Omron CX-Programmer project NewProject (CX-Programmer 9.74)

# PLC MES_Trat: CJ2M CPU34
I/O table (CPU CJ2M-CPU34): rack 0 slot 0 CJ1W-OD232; rack 0 slot 11 CJ2M-EIP21

## Data types
TYPE Evento : STRUCT
  Ciclo : BOOL;  (* Em Ciclo Produtivo PLC->MES *)
  Estado : INT;  (* Estado Equipamento PLC->MES *)
  EquiDesabil : BOOL Dimensions=[16];  (* Equipamento Desabilitado PLC->MES *)
  FimCiclo : BOOL;  (* Finalização Ciclo PLC->MES *)
END_STRUCT END_TYPE
TYPE Ordem_Cmd : STRUCT
  AutoMES : BOOL;  (* Autorização MES MES->PLC *)
  QtdFaltaOF : UDINT;  (* Quantidade Em Falta OF *)
  ProdExecMaquina : UDINT;  (* Produção Executada Máquina *)
END_STRUCT END_TYPE
TYPE Ordem : STRUCT
  Ordem : DINT;  (* OF_OM MES->PLC *)
  Sinalizacao : BOOL;
  ProdExpect : UDINT;  (* Produção Expectável MES->PLC *)
  ProdExecOrdem : UDINT;  (* Produção Executada Ordem MES->PLC *)
END_STRUCT END_TYPE
TYPE InfoAux : STRUCT
  Cliente : WORD Dimensions=[50];  (* Cliente (string) MES->PLC *)
  Artigo : WORD Dimensions=[50];  (* Artigo (string) MES->PLC *)
  Encomenda : WORD Dimensions=[50];  (* Encomenda (string) MES->PLC *)
  QtdEncom : UDINT;  (* Quantidade Encomenda MES->PLC *)
  QtdReal : UDINT;  (* Quantidade Real MES->PLC *)
  NomeReceita : WORD Dimensions=[50];  (* Nome Receita (string) MES->PLC *)
  DataExpedic : WORD Dimensions=[4];  (* Data Expedição (string) MES->PLC *)
END_STRUCT END_TYPE
TYPE BStep : STRUCT  (* Batch Load/Exec Steps defenition *)
  Func : DWORD;  (* Function *)
  Param01 : DWORD;
  Param02 : DWORD;
END_STRUCT END_TYPE
TYPE BatchLoad : STRUCT
  InfoAux : InfoAux;
  Ordem : DINT;  (* Ordem MES->PLC *)
  Chk : WORD;  (* CheckSum MES->PLC *)
  Steps : BStep Dimensions=[12];  (* Steps MES->PLC *)
END_STRUCT END_TYPE
TYPE BatchExec : STRUCT
  Steps : BStep Dimensions=[12];  (* PLC->MES *)
END_STRUCT END_TYPE
TYPE RStep : STRUCT  (* Batch Real Step defenition *)
  Active : BOOL;
  Value01 : DWORD;
  Value02 : DWORD;
END_STRUCT END_TYPE
TYPE BatchReal : STRUCT
  Heat : RStep;  (* PLC->MES *)
  Inje : RStep;  (* PLC->MES *)
  Dedu : RStep;  (* PLC->MES *)
  Tumb : RStep;  (* PLC->MES *)
  Load : RStep;  (* PLC->MES *)
  Unload : RStep;  (* PLC->MES *)
END_STRUCT END_TYPE
TYPE s_of_totais : STRUCT  (* Totais produzidos e a produzir de uma OF *)
  tt_global : UDINT;  (* Total a produzir na OF *)
  tt_falta : UDINT;  (* Total que falta produzir na OF *)
  tt_produzir : UDINT;  (* Total a produzir na maquina no batch *)
  tt_cestos : UDINT;  (* Total de cestos a produzir na OF *)
END_STRUCT END_TYPE
TYPE s_of_cliente : STRUCT  (* Dados do cliente de uma OF *)
  Cliente : WORD Dimensions=[50];
  Artigo : WORD Dimensions=[50];
  Encomenda : WORD Dimensions=[50];
  QtdEncomenda : UDINT;
  QtdReal : UDINT;
  DataExpedicao : WORD Dimensions=[4];
  NomeReceita : WORD Dimensions=[50];
  nome : WORD Dimensions=[25];
  data : WORD Dimensions=[10];
  produto : WORD Dimensions=[20];
  prg_on : WORD Dimensions=[5];
  n_enc : WORD Dimensions=[10];
  n_of : WORD Dimensions=[10];
  n_lt : WORD Dimensions=[10];
  rsv2 : INT Dimensions=[10];
END_STRUCT END_TYPE
TYPE s_of_pss : STRUCT  (* Passo individual do programa a executar *)
  f : INT;  (* Função *)
  p1 : INT;  (* Parametro 1 *)
  p2 : REAL;  (* Parametro 2 *)
  tt : REAL;  (* Totalizador *)
  uni : INT;  (* Unidade *)
  b0 : BOOL;  (* Bit - É função *)
  b1 : BOOL;  (* Bit - É produto *)
  b2 : BOOL;  (* Bit - Tem tempo *)
  b3 : BOOL;  (* Bit - Tem quantidade *)
  b4 : BOOL;  (* Bit - Tem temperatura *)
  tt_inv : REAL;  (* Contagem Inversa *)
END_STRUCT END_TYPE
TYPE s_of_prg : STRUCT  (* Programa a ser executado *)
  pss : s_of_pss Dimensions=[12];  (* Passos do programa a executar *)
END_STRUCT END_TYPE
TYPE s_of : STRUCT  (* Ordem de fabrico *)
  cliente : s_of_cliente;  (* Cliente da OF *)
  totais : s_of_totais;  (* Totais da OF *)
  dados : BOOL;  (* OF com valores *)
  online : BOOL;  (* Ordem com dados para funcionar online *)
  rep : BOOL;  (* OF/Lote reprocessado *)
  of_del : BOOL;  (* Apagar OF *)
  sel_cestos_rolhas : BOOL;  (* Botão de Selecção entre inserção de número de rolhas e número de cestos a produzir *)
  nprg_off : INT;  (* Numero do programa offline *)
  prg : s_of_prg;  (* Programa *)
END_STRUCT END_TYPE
TYPE Passos : STRUCT
  f : INT;
  p1 : INT;
  p2 : REAL;
END_STRUCT END_TYPE
TYPE ReceitaMaq : STRUCT
  Step : Passos Dimensions=[12];
END_STRUCT END_TYPE
TYPE s_Steps : STRUCT
  f : INT;  (* Função *)
  p1 : INT;  (* Parametro 1 *)
  p2 : REAL;  (* Parametro 2 *)
END_STRUCT END_TYPE
TYPE s_Step : STRUCT
  f : INT;  (* Função *)
  p1 : INT;  (* Parametro 1 *)
  p2 : REAL;  (* Parametro 2 *)
  No : INT;  (* Numero do Passo *)
END_STRUCT END_TYPE
TYPE s_Estado : STRUCT
  Ciclo : BOOL;  (* Em ciclo produtivo *)
  FimCiclo : BOOL;  (* Finalização ciclo *)
  Estado : BOOL;  (* Estado equipamento *)
  FimTratamento : BOOL;  (* Tratamento Finalizado *)
  OF_Carregada : BOOL;  (* Ordem carregada para máquina *)
  Avaria : BOOL;  (* Máquina em Avaria *)
  Com_OF : BOOL;  (* Máquina com OF carregada *)
  FalhaInjeProd : BOOL;  (* Falta de injeção de produto *)
  FalhaAquecim : BOOL;  (* Falha de aquecimento *)
  AvariaTermicos : BOOL;  (* Avaria de térmicos *)
  TratAbortado : BOOL;  (* Tratamento abortado pelo operador *)
  FalhaEnergia : BOOL;  (* Falha energia *)
  NivelProdBaixo : BOOL;  (* Nível produto químico no depósito baixo *)
  Manual : BOOL;  (* modo manual *)
  Emergencia : BOOL;  (* Paragem Emergência *)
END_STRUCT END_TYPE
TYPE s_produtos : STRUCT
  CodMES : WORD Dimensions=[4];
  CodPLC : INT;
END_STRUCT END_TYPE
TYPE M1_Param : STRUCT  (* Parametros do passo *)
  Manual : BOOL;  (* Espera por confirmação manual do operador *)
  Auto : BOOL;  (* Avança automáticamente *)
  P1 : BOOL;  (* Produto 1 *)
  P2 : BOOL;  (* Produto 2 *)
  P3 : BOOL;  (* Produto 3 *)
  P4 : BOOL;  (* Produto 4 *)
  DEDU : BOOL;  (* Asperação (Blower) *)
  HEAT : BOOL;  (* Aquecimento (Heater) *)
  TUMB : BOOL;  (* Rotação (Speed) *)
  LOAD : BOOL;  (* Carga *)
  UNLO : BOOL;  (* Descarga (unload) *)
  Reserva : BOOL;
  End : BOOL;
  CalTemp : BOOL;  (* Calor por Temperatura *)
  Cool : BOOL;  (* Arrefecimento *)
END_STRUCT END_TYPE
TYPE M1_ParamProd : STRUCT  (* Parametros produtos *)
  DoseRate : BOOL;  (* por Dosagem g/m *)
  Qtd : BOOL;  (* por Quantidade q *)
  Time : BOOL;  (* poe Tempo mm:ss *)
  Cycles : BOOL;  (* por Ciclos *)
END_STRUCT END_TYPE
TYPE M1_Step : STRUCT  (* Passo da Receita *)
  Parametros : M1_Param;  (* Parametros do Passo *)
  ParamProdutos : M1_ParamProd Dimensions=[4];
  Temperatura : INT;  (* Valor da Temperatura *)
  Velocidade : INT;  (* Valor Velocidade Rotação (%) *)
  P1 : INT;  (* Valor Produto 1 *)
  P2 : INT;  (* Valor Produto 2 *)
  P3 : INT;  (* Valor Produto 3 *)
  P4 : BOOL;  (* Valor do Produto 4 *)
  Tempo : BOOL;  (* Tempo (mm:ss) *)
  Reserva : INT;
  P1_TOff_TOn : INT;  (* TOff/TON P1 *)
  P2_TOff_TOn : INT;  (* TOff/TON P2 *)
  P3_TOff_TOn : INT;  (* TOff/TON P3 *)
  P4_TOff_TOn : INT;  (* TOff/TON P4 *)
END_STRUCT END_TYPE
TYPE s_Controlo : STRUCT
  Mannual : BOOL;
  Auto : BOOL;
  P1 : BOOL;
  P2 : BOOL;
  P3 : BOOL;
  P4 : BOOL;
  Aspiracao : BOOL;
  Aquecimento : BOOL;
  Rotacao : BOOL;
  Carga : BOOL;
  Descarga : BOOL;
  Reserva1 : BOOL;
  Fim : BOOL;
  CalorPorTemperatura : BOOL;
  Arrefecimento : BOOL;
  Reserva2 : BOOL;
  Ctrl_P1 : s_CtrlProduto;
  Ctrl_P2 : s_CtrlProduto;
  Ctrl_P3 : s_CtrlProduto;
  Ctrl_P4 : BOOL;
END_STRUCT END_TYPE
TYPE s_CtrlProduto : STRUCT  (* Bits controlo produto *)
  DoseRate : BOOL;
  Qtd : BOOL;
  Time : BOOL;
  Cycles : BOOL;
END_STRUCT END_TYPE
TYPE s_StepRcpMaq1 : STRUCT  (* Receita máquina 1 *)
  Control : s_Controlo;
  Temperatura : UINT;
  Velocidade : UINT;
  ValorProduto : UINT;  (* Valor do Produto a Injetar (minutos/segundos) *)
  Tempo : UINT;  (* Tempo em segundos (minutos/segundos) *)
END_STRUCT END_TYPE
TYPE s_Evento : STRUCT
  HeartBeat : INT;  (* Heart Beat Maquina *)
  TSemHB : INT;  (* Tempo Sem Heart Beat *)
END_STRUCT END_TYPE
TYPE MqDL : STRUCT  (* 'All the mid-branches are substituted bu ".sub_Fcn."' *)
  Ordem : DINT;
  Ordem_BL : DINT;
  ProdExpect : UDINT;
  ProdEecOrdem : UDINT;
  QtdEncom : UDINT;
  QtdReal : UDINT;
  QtdEncom_BL : UDINT;
  QtdReal_BL : UDINT;
  Sinalizacao : BOOL Dimensions=[32];
  Cliente : WORD Dimensions=[50];
  Artigo : WORD Dimensions=[50];
  Encomenda : WORD Dimensions=[50];
  NomeReceita : WORD Dimensions=[50];
  Cliente_BL : WORD Dimensions=[50];
  Artigo_BL : WORD Dimensions=[50];
  Encomenda_BL : WORD Dimensions=[50];
  NomeReceita_BL : WORD Dimensions=[50];
  DataExpedic_BL : WORD Dimensions=[4];
  DataExpedic : WORD Dimensions=[4];
  Steps_BL : BStep Dimensions=[12];
END_STRUCT END_TYPE
TYPE MqRT : STRUCT  (* 'All the mid-branches are substituted bu ".sub_Fcn."' *)
  Ciclo : BOOL;
  Estado : INT;
  EquiDesabil : BOOL Dimensions=[16];
  FimCiclo : BOOL Dimensions=[16];
  AutoMes : BOOL Dimensions=[16];
  QtdFaltaOF : UDINT;
  ProExecOrdem : UDINT;
  Chk : WORD;
  Temperatura : UINT;
  BatchReal : BatchReal;
  Destination : UINT;
END_STRUCT END_TYPE

## Global symbols (name address type ; comment)
BatchReal_Maq01 E0_23050 STRUCT s_Steps
BatchReal_Maq02 E0_23150 STRUCT s_Steps
BatchReal_Maq03 E0_23250 STRUCT s_Steps
BatchReal_Maq04 E0_23350 STRUCT s_Steps
BatchReal_Maq05 E0_23450 STRUCT s_Steps
BatchReal_Maq06 E0_23550 STRUCT s_Steps
BatchReal_Maq07 E0_23650 STRUCT s_Steps
BatchReal_Maq08 E0_23750 STRUCT s_Steps
BatchReal_Maq09 E0_23850 STRUCT s_Steps
BatchReal_Maq10 E0_23950 STRUCT s_Steps
BatchReal_Maq11 E0_24050 STRUCT s_Steps
CHK_M01 D12290 WORD
CHK_M02 D12293 WORD
CHK_M03 D12296 WORD
CHK_M04 D12299 WORD
CHK_M05 D12302 WORD
CHK_M06 D12305 WORD
CHK_M07 D12308 WORD
CHK_M08 D12311 WORD
CHK_M09 D12314 WORD
CHK_M10 D12317 WORD
CHK_M11 D12320 WORD
CopyStps CopySteps
CopyStps09 CopySteps
CopyStps10 CopySteps
CopyStps11 CopySteps
CopyStps2 CopySteps
CopyStps3 CopySteps
CopyStps4 CopySteps
CopyStps5 CopySteps
CopyStps6 CopySteps
CopyStps7 CopySteps
CopyStps8 CopySteps
Estado_Maq01 E0_23057 STRUCT s_Estado
Estado_Maq02 E0_23157 STRUCT s_Estado
Estado_Maq03 E0_23257 STRUCT s_Estado
Estado_Maq04 E0_23357 STRUCT s_Estado
Estado_Maq05 E0_23457 STRUCT s_Estado
Estado_Maq06 E0_23557 STRUCT s_Estado
Estado_Maq07 E0_23657 STRUCT s_Estado
Estado_Maq08 E0_23757 STRUCT s_Estado
Estado_Maq09 E0_23857 STRUCT s_Estado
Estado_Maq10 E0_23957 STRUCT s_Estado
Estado_Maq11 E0_24057 STRUCT s_Estado
HB_M01 D12288 INT
HB_M02 D12291 INT
HB_M03 D12294 INT
HB_M04 D12297 INT
HB_M05 D12300 INT
HB_M06 D12303 INT
HB_M07 D12306 INT
HB_M08 D12309 INT
HB_M09 D12312 INT
HB_M10 D12315 INT
HB_M11 D12318 INT
M1_Tsfr_Rqst E0_25100.00 BOOL
M2_Tsfr_Rqst E0_25100.01 BOOL
M3_Tsfr_Rqst E0_25100.02 BOOL
M4_Tsfr_Rqst E0_25100.03 BOOL
M5_Tsfr_Rqst E0_25100.04 BOOL
M6_Tsfr_Rqst E0_25100.05 BOOL
MQ01_InfoAuxMq D15000 STRUCT InfoAux  ; InfoAux da receita na máquina
MQ02_InfoAuxMq D15250 STRUCT InfoAux  ; InfoAux da receita na máquina
MQ03_InfoAuxMq D15500 STRUCT InfoAux  ; InfoAux da receita na máquina
MQ04_InfoAuxMq D15750 STRUCT InfoAux  ; InfoAux da receita na máquina
MQ05_InfoAuxMq D16000 STRUCT InfoAux  ; InfoAux da receita na máquina
MQ06_InfoAuxMq D16250 STRUCT InfoAux  ; InfoAux da receita na máquina
MQ07_InfoAuxMq D16500 STRUCT InfoAux  ; InfoAux da receita na máquina
MQ08_InfoAuxMq D16750 STRUCT InfoAux  ; InfoAux da receita na máquina
MQ09_InfoAuxMq D17000 STRUCT InfoAux  ; InfoAux da receita na máquina
MQ10_InfoAuxMq D17250 STRUCT InfoAux  ; InfoAux da receita na máquina
MQ11_InfoAuxMq D17500 STRUCT InfoAux  ; InfoAux da receita na máquina
MaqDL_01 D5120 STRUCT MqDL
MaqDL_02 D5618 STRUCT MqDL
MaqDL_03 D6116 STRUCT MqDL
MaqDL_04 D6614 STRUCT MqDL
MaqDL_05 D7112 STRUCT MqDL
MaqDL_06 D7610 STRUCT MqDL
MaqDL_07 D8108 STRUCT MqDL
MaqDL_08 D8606 STRUCT MqDL
MaqDL_09 D9104 STRUCT MqDL
MaqDL_10 D9602 STRUCT MqDL
MaqDL_11 D10100 STRUCT MqDL
MaqRT_01 D0 STRUCT MqRT
MaqRT_02 D42 STRUCT MqRT
MaqRT_03 D84 STRUCT MqRT
MaqRT_04 D126 STRUCT MqRT
MaqRT_05 D168 STRUCT MqRT
MaqRT_06 D210 STRUCT MqRT
MaqRT_07 D252 STRUCT MqRT
MaqRT_08 D294 STRUCT MqRT
MaqRT_09 D336 STRUCT MqRT
MaqRT_10 D378 STRUCT MqRT
MaqRT_11 D420 STRUCT MqRT
MaqRcpNetIN_01 E0_10000 STRUCT s_of
MaqRcpNetIN_02 E0_11000 STRUCT s_of
MaqRcpNetIN_03 E0_12000 STRUCT s_of
MaqRcpNetIN_04 E0_13000 STRUCT s_of
MaqRcpNetIN_05 E0_14000 STRUCT s_of
MaqRcpNetIN_06 E0_15000 STRUCT s_of
MaqRcpNetIN_07 E0_16000 STRUCT s_of
MaqRcpNetIN_08 E0_17000 STRUCT s_of
MaqRcpNetIN_09 E0_18000 STRUCT s_of
MaqRcpNetIN_10 E0_19000 STRUCT s_of
MaqRcpNetIN_11 E0_20000 STRUCT s_of
MaqRcpNet_01 E0_0 STRUCT s_of
MaqRcpNet_02 E0_1000 STRUCT s_of
MaqRcpNet_03 E0_2000 STRUCT s_of
MaqRcpNet_04 E0_3000 STRUCT s_of
MaqRcpNet_05 E0_4000 STRUCT s_of
MaqRcpNet_06 E0_5000 STRUCT s_of
MaqRcpNet_07 E0_6000 STRUCT s_of
MaqRcpNet_08 E0_7000 STRUCT s_of
MaqRcpNet_09 E0_8000 STRUCT s_of
MaqRcpNet_10 E0_9000 STRUCT s_of
MaqRcpNet_11 E0_21000 STRUCT s_of
Mq09_CRC_Calc RecipeCRC
Mq10_CRC_Calc RecipeCRC
Mq11_CRC_Calc RecipeCRC
Mq1_CRC_Calc RecipeCRC
Mq2_CRC_Calc RecipeCRC
Mq3_CRC_Calc RecipeCRC
Mq4_CRC_Calc RecipeCRC
Mq5_CRC_Calc RecipeCRC
Mq6_CRC_Calc RecipeCRC
Mq7_CRC_Calc RecipeCRC
Mq8_CRC_Calc RecipeCRC
PLC_MES PLC_to_MES
PLC_MES09 PLC_to_MES
PLC_MES10 PLC_to_MES
PLC_MES11 PLC_to_MES
PLC_MES2 PLC_to_MES
PLC_MES3 PLC_to_MES
PLC_MES4 PLC_to_MES
PLC_MES5 PLC_to_MES
PLC_MES6 PLC_to_MES
PLC_MES7 PLC_to_MES
PLC_MES8 PLC_to_MES
Produtos H0 STRUCT[13] s_produtos
RcpTrans RecipeTranslate
RcpTrans09 RecipeTranslate
RcpTrans10 RecipeTranslate
RcpTrans11 RecipeTranslate
RcpTrans2 RecipeTranslate
RcpTrans3 RecipeTranslate
RcpTrans4 RecipeTranslate
RcpTrans5 RecipeTranslate
RcpTrans6 RecipeTranslate
RcpTrans7 RecipeTranslate
RcpTrans8 RecipeTranslate
RcpTst RecipeTst
RcpTst09 RecipeTst
RcpTst10 RecipeTst
RcpTst11 RecipeTst
RcpTst2 RecipeTst
RcpTst3 RecipeTst
RcpTst4 RecipeTst
RcpTst5 RecipeTst
RcpTst6 RecipeTst
RcpTst7 RecipeTst
RcpTst8 RecipeTst
ReceitaMaqOK_01 E0_23048.00 BOOL
ReceitaMaqOK_02 E0_23148.00 BOOL
ReceitaMaqOK_03 E0_23248.00 BOOL
ReceitaMaqOK_04 E0_23348.00 BOOL
ReceitaMaqOK_05 E0_23448.00 BOOL
ReceitaMaqOK_06 E0_23548.00 BOOL
ReceitaMaqOK_07 E0_23648.00 BOOL
ReceitaMaqOK_08 E0_23748.00 BOOL
ReceitaMaqOK_09 E0_23848.00 BOOL
ReceitaMaqOK_10 E0_23948.00 BOOL
ReceitaMaqOK_11 E0_24048.00 BOOL
ReceitaMaq_01 E0_23000 STRUCT[12] Passos
ReceitaMaq_02 E0_23100 STRUCT[12] Passos
ReceitaMaq_03 E0_23200 STRUCT[12] Passos
ReceitaMaq_04 E0_23300 STRUCT[12] Passos
ReceitaMaq_05 E0_23400 STRUCT[12] Passos
ReceitaMaq_06 E0_23500 STRUCT[12] Passos
ReceitaMaq_07 E0_23600 STRUCT[12] Passos
ReceitaMaq_08 E0_23700 STRUCT[12] Passos
ReceitaMaq_09 E0_23800 STRUCT[12] Passos
ReceitaMaq_10 E0_23900 STRUCT[12] Passos
ReceitaMaq_11 E0_24000 STRUCT[12] Passos
Send_M7 _CPU010_SendData
TSemHB_M01 D12289 INT
TSemHB_M02 D12292 INT
TSemHB_M03 D12295 INT
TSemHB_M04 D12298 INT
TSemHB_M05 D12301 INT
TSemHB_M06 D12304 INT
TSemHB_M07 D12307 INT
TSemHB_M08 D12310 INT
TSemHB_M09 D12313 INT
TSemHB_M10 D12316 INT
TSemHB_M11 D12319 INT
Teperatura_Maq01 E0_23055 INT
Teperatura_Maq02 E0_23155 INT
Teperatura_Maq03 E0_23255 INT
Teperatura_Maq04 E0_23355 INT
Teperatura_Maq05 E0_23455 INT
Teperatura_Maq06 E0_23555 INT
Teperatura_Maq07 E0_23655 INT  ; ~
Teperatura_Maq08 E0_23755 INT
Teperatura_Maq09 E0_23855 INT
Teperatura_Maq10 E0_23955 INT
Teperatura_Maq11 E0_24055 INT
Transfer FIFO
TranspDest_Maq01 E0_23056 UINT
TranspDest_Maq02 E0_23156 UINT
TranspDest_Maq03 E0_23256 UINT
TranspDest_Maq04 E0_23356 UINT
TranspDest_Maq05 E0_23456 UINT
TranspDest_Maq06 E0_23556 UINT
TranspDest_Maq07 E0_23656 UINT
TranspDest_Maq08 E0_23756 UINT
TranspDest_Maq09 E0_23856 UINT
TranspDest_Maq10 E0_23956 UINT
TranspDest_Maq11 E0_24056 UINT
out_M_A_SinAmarelo 0.01 BOOL  ; Sinalizador amarelo
out_M_A_SinAzul 0.04 BOOL  ; Sinalizador azul
out_M_A_SinBranco 0.02 BOOL  ; Sinalizador branco
out_M_A_SinVerde 0.03 BOOL  ; Sinalizador verde
out_M_A_SinVermelho 0.00 BOOL  ; Sinalizador vermelho
out_M_B_SinAmarelo 0.06 BOOL  ; Sinalizador amarelo
out_M_B_SinAzul 0.09 BOOL  ; Sinalizador azul
out_M_B_SinBranco 0.07 BOOL  ; Sinalizador branco
out_M_B_SinVerde 0.08 BOOL  ; Sinalizador verde
out_M_B_SinVermelho 0.05 BOOL  ; Sinalizador vermelho
out_M_C_SinAmarelo 0.11 BOOL  ; Sinalizador amarelo
out_M_C_SinAzul 0.14 BOOL  ; Sinalizador azul
out_M_C_SinBranco 0.12 BOOL  ; Sinalizador branco
out_M_C_SinVerde 0.13 BOOL  ; Sinalizador verde
out_M_C_SinVermelho 0.10 BOOL  ; Sinalizador vermelho
out_M_D_SinAmarelo 1.00 BOOL  ; Sinalizador amarelo
out_M_D_SinAzul 1.03 BOOL  ; Sinalizador azul
out_M_D_SinBranco 1.01 BOOL  ; Sinalizador branco
out_M_D_SinVerde 1.02 BOOL  ; Sinalizador verde
out_M_D_SinVermelho 0.15 BOOL  ; Sinalizador vermelho
tst_str W0 STRING[200]

## Program NewProgram1 (cyclic task 0)
Local symbols
CNT_HB3 W66 UINT
Dummy W1.00 BOOL
EmpyStr W62 STRING[2]
Err_CHK_MQ01 W301.00 BOOL
Err_CHK_MQ02 W301.01 BOOL
Err_CHK_MQ03 W301.02 BOOL
Err_CHK_MQ04 W301.03 BOOL
Err_CHK_MQ05 W301.04 BOOL
Err_CHK_MQ06 W301.05 BOOL
Err_CHK_MQ07 W301.06 BOOL  ; ~
Err_CHK_MQ08 W301.07 BOOL
Err_CHK_MQ09 W301.08 BOOL
Err_CHK_MQ10 W301.09 BOOL
Err_CHK_MQ11 W301.10 BOOL
HB_Atraso W65 UINT
IP W64 UINT
LampShift W67 UINT
M08_Enable W32.11 BOOL
M09_Enable W32.12 BOOL
M10_Enable W32.03 BOOL
M11_Enable W35.08 BOOL
M1_Enable W32.02 BOOL
M2_Enable W32.04 BOOL
M3_Enable W32.05 BOOL
M4_Enable W32.06 BOOL
M5_Enable W32.07 BOOL
M6_Enable W32.08 BOOL
M7_Enable W32.09 BOOL
M7_Err W102 WORD
M7e8_Bussy W101.00 BOOL  ; ~
M8_Enable W32.10 BOOL
MQ1_CRC W0 WORD
Mestre_01 W34.15 BOOL
Mestre_02 W35.00 BOOL
Mestre_03 W35.01 BOOL
P_Ciclo W35.06 BOOL
RcpOk_M09 W30.07 BOOL
RcpOk_M1 W30.14 BOOL
RcpOk_M10 W33.06 BOOL
RcpOk_M11 W33.15 BOOL
RcpOk_M2 W29.07 BOOL
RcpOk_M3 W30.10 BOOL
RcpOk_M4 W29.04 BOOL
RcpOk_M5 W29.12 BOOL
RcpOk_M6 W29.10 BOOL
RcpOk_M7 W34.06 BOOL
RcpOk_M8 W29.14 BOOL
RcpToProduction W29.03 BOOL
RcpToProduction09 W30.06 BOOL
RcpToProduction10 W33.05 BOOL
RcpToProduction11 W33.14 BOOL
RcpToProduction2 W29.06 BOOL
RcpToProduction3 W30.09 BOOL
RcpToProduction4 W30.12 BOOL
RcpToProduction5 W34.01 BOOL
RcpToProduction6 W29.09 BOOL
RcpToProduction7 W34.05 BOOL
RcpToProduction8 W29.13 BOOL
RcpTst_Res W7.00 BOOL[16]
RcpTst_Res09 W26.00 BOOL[16]
RcpTst_Res10 W27.00 BOOL[16]
RcpTst_Res11 W28.00 BOOL[16]
RcpTst_Res2 W8.00 BOOL[16]
RcpTst_Res3 W9.00 BOOL[16]
RcpTst_Res4 W21.00 BOOL[16]
RcpTst_Res5 W22.00 BOOL[16]
RcpTst_Res6 W23.00 BOOL[16]
RcpTst_Res7 W24.00 BOOL[16]
RcpTst_Res8 W25.00 BOOL[16]
RcpTst_Res_Ok01 W300.00 BOOL
RcpTst_Res_Ok02 W300.01 BOOL
RcpTst_Res_Ok03 W300.02 BOOL
RcpTst_Res_Ok04 W300.03 BOOL
RcpTst_Res_Ok05 W300.04 BOOL
RcpTst_Res_Ok06 W300.05 BOOL
RcpTst_Res_Ok07 W300.06 BOOL
RcpTst_Res_Ok08 W300.07 BOOL
RcpTst_Res_Ok09 W300.08 BOOL
RcpTst_Res_Ok10 W300.09 BOOL
RcpTst_Res_Ok11 W300.10 BOOL
ReceitaMaqOK_7 W34.07 BOOL
Recipe_Ok W4.00 BOOL
T_SemHB_M01 W47 INT
T_SemHB_M02 W48 INT
T_SemHB_M03 W50 INT
T_SemHB_M04 W51 INT
T_SemHB_M05 W52 INT
T_SemHB_M06 W56 INT
T_SemHB_M07 W57 INT
T_SemHB_M08 W58 INT
T_SemHB_M09 W59 INT
T_SemHB_M10 W60 INT
T_SemHB_M11 W61 INT
Zero_Dint W68 DINT
bit_1s W2.00 BOOL
bit_CRC_Calc W5.00 BOOL
bit_CRC_Calc07 W34.03 BOOL
bit_CRC_Calc09 W30.00 BOOL
bit_CRC_Calc10 W33.02 BOOL
bit_CRC_Calc11 W33.11 BOOL
bit_CRC_Calc2 W6.00 BOOL
bit_CRC_Calc3 W10.00 BOOL
bit_CRC_Calc4 W11.00 BOOL
bit_CRC_Calc5 W18.11 BOOL
bit_CRC_Calc6 W19.01 BOOL
bit_CRC_Calc7 W19.07 BOOL
bit_CRC_Calc8 W19.13 BOOL
bit_CRC_Calc_End W12.00 BOOL
bit_CRC_Calc_End07 W34.04 BOOL
bit_CRC_Calc_End09 W30.01 BOOL
bit_CRC_Calc_End10 W30.15 BOOL
bit_CRC_Calc_End11 W33.08 BOOL
bit_CRC_Calc_End2 W13.00 BOOL
bit_CRC_Calc_End3 W14.00 BOOL
bit_CRC_Calc_End35 W35.04 BOOL
bit_CRC_Calc_End4 W15.00 BOOL
bit_CRC_Calc_End5 W18.12 BOOL
bit_CRC_Calc_End6 W19.02 BOOL
bit_CRC_Calc_End7 W19.08 BOOL
bit_CRC_Calc_End8 W19.14 BOOL
bit_CRC_Calc_Retry W16.00 BOOL
bit_CRC_Calc_Retry09 W30.04 BOOL
bit_CRC_Calc_Retry10 W33.03 BOOL
bit_CRC_Calc_Retry11 W33.12 BOOL
bit_CRC_Calc_Retry2 W17.00 BOOL
bit_CRC_Calc_Retry3 W18.00 BOOL
bit_CRC_Calc_Retry4 W18.01 BOOL
bit_CRC_Calc_Retry5 W18.15 BOOL
bit_CRC_Calc_Retry6 W19.05 BOOL
bit_CRC_Calc_Retry7 W19.11 BOOL
bit_CRC_Calc_Retry8 W29.01 BOOL
bit_CRC_NOK W18.02 BOOL
bit_CRC_NOK09 W30.03 BOOL
bit_CRC_NOK10 W32.01 BOOL
bit_CRC_NOK11 W33.10 BOOL
bit_CRC_NOK2 W18.03 BOOL
bit_CRC_NOK3 W18.04 BOOL  ; ~
bit_CRC_NOK4 W18.05 BOOL
bit_CRC_NOK5 W18.14 BOOL
bit_CRC_NOK6 W19.04 BOOL
bit_CRC_NOK7 W19.10 BOOL
bit_CRC_NOK8 W29.00 BOOL
bit_CRC_Ok W18.06 BOOL
bit_CRC_Ok09 W30.02 BOOL
bit_CRC_Ok10 W32.00 BOOL
bit_CRC_Ok11 W33.09 BOOL
bit_CRC_Ok2 W18.07 BOOL
bit_CRC_Ok3 W18.08 BOOL
bit_CRC_Ok4 W18.09 BOOL
bit_CRC_Ok5 W18.13 BOOL
bit_CRC_Ok6 W19.03 BOOL
bit_CRC_Ok7 W19.09 BOOL
bit_CRC_Ok8 W19.15 BOOL
bit_CRC_Ok9 W101.09 BOOL
bit_Ciclo W35.07 BOOL
bit_ComOrdem_M01 W3.00 BOOL
bit_ComOrdem_M02 W18.10 BOOL
bit_ComOrdem_M03 W19.00 BOOL
bit_ComOrdem_M04 W19.06 BOOL
bit_ComOrdem_M05 W19.12 BOOL
bit_ComOrdem_M06 W29.02 BOOL
bit_ComOrdem_M07 W30.05 BOOL
bit_ComOrdem_M08 W33.04 BOOL
bit_ComOrdem_M09 W33.13 BOOL
bit_ComOrdem_M10 W35.02 BOOL
bit_ComOrdem_M11 W35.03 BOOL
bit_LampTst W1.01 BOOL
bit_Limpa W29.05 BOOL
bit_Limpa09 W30.08 BOOL
bit_Limpa10 W33.07 BOOL
bit_Limpa11 W34.00 BOOL
bit_Limpa2 W29.08 BOOL
bit_Limpa3 W30.11 BOOL
bit_Limpa4 W30.13 BOOL
bit_Limpa5 W34.02 BOOL
bit_Limpa6 W29.11 BOOL
bit_Limpa7 W34.08 BOOL
bit_Limpa8 W29.15 BOOL
bit_M01_SinAmarelo W49.05 BOOL  ; Sinalizador amarelo . Tratamento Nº1
bit_M01_SinAzul W49.08 BOOL  ; Sinalizador azul - Tratamento Nº1
bit_M01_SinBranco W49.06 BOOL  ; Sinalizador branco - Tratamento Nº1
bit_M01_SinVerde W49.07 BOOL  ; Sinalizador verde - Tratamento Nº1
bit_M01_SinVermelho W49.04 BOOL  ; Sinalizador vermelho - Tratamento Nº1
bit_M02_SinAmarelo W49.10 BOOL  ; Sinalizador amarelo . Tratamento Nº2
bit_M02_SinAzul W49.13 BOOL  ; Sinalizador azul - Tratamento Nº2
bit_M02_SinBranco W49.11 BOOL  ; Sinalizador branco - Tratamento Nº2
bit_M02_SinVerde W49.12 BOOL  ; Sinalizador verde - Tratamento Nº2
bit_M02_SinVermelho W49.09 BOOL  ; Sinalizador vermelho - Tratamento Nº2
bit_M03_SinAmarelo W49.15 BOOL  ; Sinalizador amarelo . Tratamento Nº3
bit_M03_SinAzul W53.02 BOOL  ; Sinalizador azul - Tratamento Nº3
bit_M03_SinBranco W53.00 BOOL  ; Sinalizador branco - Tratamento Nº3
bit_M03_SinVerde W53.01 BOOL  ; Sinalizador verde - Tratamento Nº3
bit_M03_SinVermelho W49.14 BOOL  ; Sinalizador vermelho - Tratamento Nº3
bit_M04_SinAmarelo W53.04 BOOL  ; Sinalizador amarelo . Tratamento Nº4
bit_M04_SinAzul W53.07 BOOL  ; Sinalizador azul - Tratamento Nº4
bit_M04_SinBranco W53.05 BOOL  ; Sinalizador branco - Tratamento Nº4
bit_M04_SinVerde W53.06 BOOL  ; Sinalizador verde - Tratamento Nº4
bit_M04_SinVermelho W53.03 BOOL  ; Sinalizador vermelho - Tratamento Nº4
bit_M05_SinAmarelo W53.09 BOOL  ; Sinalizador amarelo . Tratamento Nº5
bit_M05_SinAzul W53.12 BOOL  ; Sinalizador azul - Tratamento Nº5
bit_M05_SinBranco W53.10 BOOL  ; Sinalizador branco - Tratamento Nº5
bit_M05_SinVerde W53.11 BOOL  ; Sinalizador verde - Tratamento Nº5
bit_M05_SinVermelho W53.08 BOOL  ; Sinalizador vermelho - Tratamento Nº5
bit_M06_SinAmarelo W53.14 BOOL  ; Sinalizador amarelo . Tratamento Nº6
bit_M06_SinAzul W54.01 BOOL  ; Sinalizador azul - Tratamento Nº6
bit_M06_SinBranco W53.15 BOOL  ; Sinalizador branco - Tratamento Nº6
bit_M06_SinVerde W54.00 BOOL  ; Sinalizador verde - Tratamento Nº6
bit_M06_SinVermelho W53.13 BOOL  ; Sinalizador vermelho - Tratamento Nº6
bit_M07_SinAmarelo W54.03 BOOL  ; Sinalizador amarelo . Tratamento Nº7
bit_M07_SinAzul W54.06 BOOL  ; Sinalizador azul - Tratamento Nº7
bit_M07_SinBranco W54.04 BOOL  ; Sinalizador branco - Tratamento Nº7
bit_M07_SinVerde W54.05 BOOL  ; Sinalizador verde - Tratamento Nº7
bit_M07_SinVermelho W54.02 BOOL  ; Sinalizador vermelho - Tratamento Nº7
bit_M08_SinAmarelo W54.08 BOOL  ; Sinalizador amarelo . Tratamento Nº8
bit_M08_SinAzul W54.11 BOOL  ; Sinalizador azul - Tratamento Nº8
bit_M08_SinBranco W54.09 BOOL  ; Sinalizador branco - Tratamento Nº8
bit_M08_SinVerde W54.10 BOOL  ; Sinalizador verde - Tratamento Nº8
bit_M08_SinVermelho W54.07 BOOL  ; Sinalizador vermelho - Tratamento Nº8
bit_M09_SinAmarelo W54.13 BOOL  ; Sinalizador amarelo . Tratamento Nº9
bit_M09_SinAzul W55.00 BOOL  ; Sinalizador azul - Tratamento Nº9
bit_M09_SinBranco W54.14 BOOL  ; Sinalizador branco - Tratamento Nº9
bit_M09_SinVerde W54.15 BOOL  ; Sinalizador verde - Tratamento Nº9
bit_M09_SinVermelho W54.12 BOOL  ; Sinalizador vermelho - Tratamento Nº9
bit_M10_SinAmarelo W55.02 BOOL  ; Sinalizador amarelo . Tratamento Nº10
bit_M10_SinAzul W55.05 BOOL  ; Sinalizador azul - Tratamento Nº10
bit_M10_SinBranco W55.03 BOOL  ; Sinalizador branco - Tratamento Nº10
bit_M10_SinVerde W55.04 BOOL  ; Sinalizador verde - Tratamento Nº10
bit_M10_SinVermelho W55.01 BOOL  ; Sinalizador vermelho - Tratamento Nº10
bit_M11_SinAmarelo W55.07 BOOL  ; Sinalizador amarelo . Tratamento Nº11
bit_M11_SinAzul W55.10 BOOL  ; Sinalizador azul - Tratamento Nº11
bit_M11_SinBranco W55.08 BOOL  ; Sinalizador branco - Tratamento Nº11
bit_M11_SinVerde W55.09 BOOL  ; Sinalizador verde - Tratamento Nº11
bit_M11_SinVermelho W55.06 BOOL  ; Sinalizador vermelho - Tratamento Nº11
bit_Maq01_ComErr W32.13 BOOL
bit_Maq02_ComErr W32.14 BOOL
bit_Maq03_ComErr W32.15 BOOL
bit_Maq04_ComErr W33.00 BOOL
bit_Maq05_ComErr W33.01 BOOL
bit_Maq06_ComErr W34.09 BOOL
bit_Maq07_ComErr W34.10 BOOL
bit_Maq08_ComErr W34.11 BOOL
bit_Maq09_ComErr W34.12 BOOL
bit_Maq10_ComErr W34.13 BOOL
bit_Maq11_ComErr W34.14 BOOL
bit_RcpTst_M01 W101.02 BOOL
bit_RcpTst_M02 W101.03 BOOL
bit_RcpTst_M03 W101.04 BOOL
bit_RcpTst_M04 W101.05 BOOL
bit_RcpTst_M05 W101.01 BOOL
bit_RcpTst_M06 W101.06 BOOL
bit_RcpTst_M07 W101.07 BOOL
bit_RcpTst_M08 W101.08 BOOL
bit_RcpTst_M09 W101.10 BOOL
bit_RcpTst_M10 W101.11 BOOL
bit_RcpTst_M11 W101.12 BOOL
cli D6839 STRING[100]
cli_1 D6639 STRING[100]
memAlrmHB W35.05 BOOL
memHB_M09 W44 INT
memHB_M1 W36 INT
memHB_M10 W45 INT
memHB_M11 W46 INT
memHB_M2 W37 INT
memHB_M3 W38 INT
memHB_M4 W39 INT
memHB_M5 W40 INT
memHB_M6 W41 INT
memHB_M7 W42 INT
memHB_M8 W43 INT
tmpMMSS W31 CHANNEL
tmpTemper W500 INT
tmp_TSemHB_M01 W204 INT
tmp_TSemHB_M02 W206 INT
tmp_TSemHB_M03 W208 INT
tmp_TSemHB_M04 W210 INT
tmp_TSemHB_M05 W212 INT
tmp_TSemHB_M06 W214 INT
tmp_TSemHB_M07 W216 INT
tmp_TSemHB_M08 W218 INT
tmp_TSemHB_M09 W220 INT
tmp_TSemHB_M10 W222 INT
tmp_TSemHB_M11 W224 INT
tst_crc W20 WORD

### Section INI

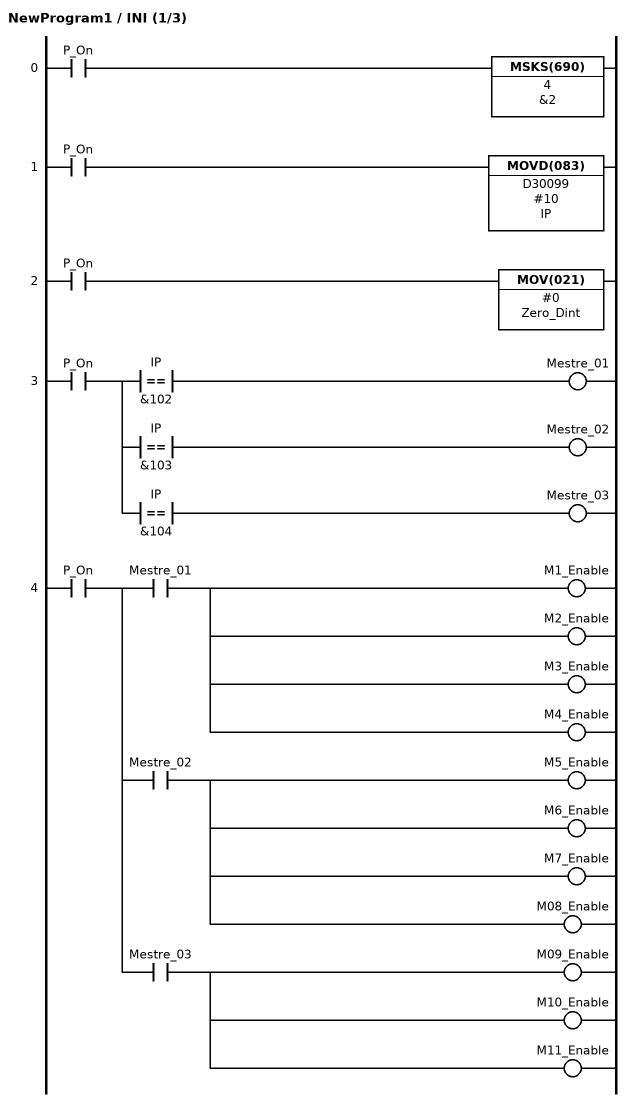
; rung 0
LD P_On
MSKS(690) 4 &2
; rung 1
LD P_On
MOVD(083) D30099 #10 IP
; rung 2
LD P_On
MOV(021) #0 Zero_Dint
; rung 3
LD P_On
OUT TR0
AND=(300) IP &102
OUT Mestre_01
LD TR0
AND=(300) IP &103
OUT Mestre_02
LD TR0
AND=(300) IP &104
OUT Mestre_03
; rung 4
LD P_On
OUT TR0
AND Mestre_01
OUT M1_Enable
OUT M2_Enable
OUT M3_Enable
OUT M4_Enable
LD TR0
AND Mestre_02
OUT M5_Enable
OUT M6_Enable
OUT M7_Enable
OUT M08_Enable
LD TR0
AND Mestre_03
OUT M09_Enable
OUT M10_Enable
OUT M11_Enable

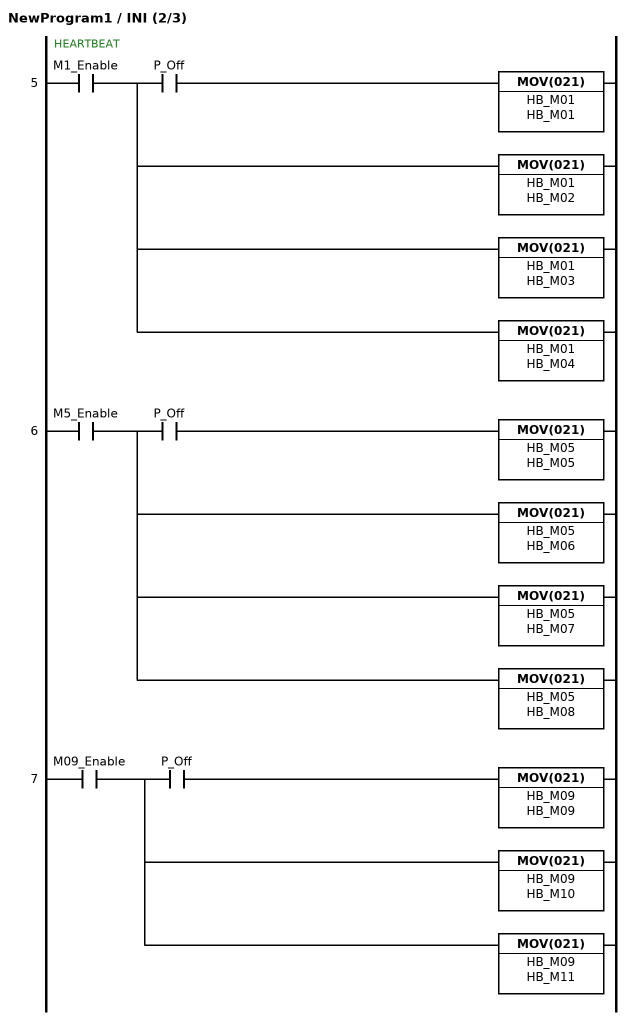
; rung 5: HEARTBEAT
LD M1_Enable
OUT TR0
AND P_Off
MOV(021) HB_M01 HB_M01
LD TR0
MOV(021) HB_M01 HB_M02
MOV(021) HB_M01 HB_M03
MOV(021) HB_M01 HB_M04
; rung 6
LD M5_Enable
OUT TR0
AND P_Off
MOV(021) HB_M05 HB_M05
LD TR0
MOV(021) HB_M05 HB_M06
MOV(021) HB_M05 HB_M07
MOV(021) HB_M05 HB_M08
; rung 7
LD M09_Enable
OUT TR0
AND P_Off
MOV(021) HB_M09 HB_M09
LD TR0
MOV(021) HB_M09 HB_M10
MOV(021) HB_M09 HB_M11

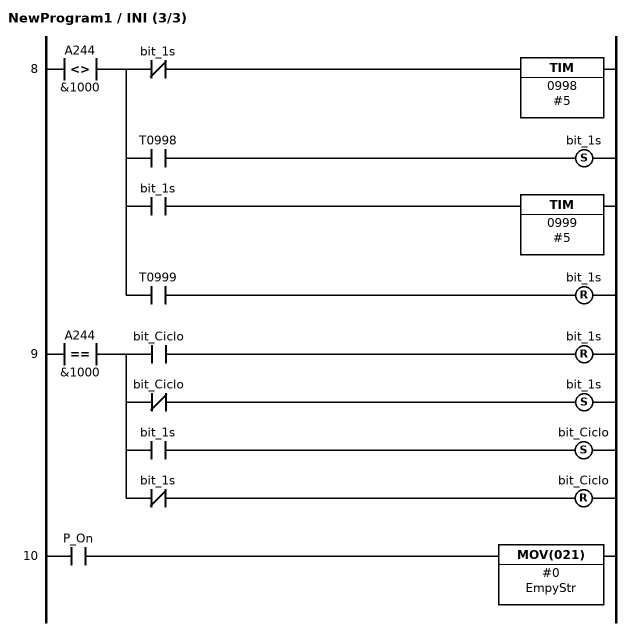
; rung 8
LD<>(305) A244 &1000
OUT TR0
ANDNOT bit_1s
TIM 0998 #5
LD TR0
AND T0998
SET bit_1s
LD TR0
AND bit_1s
TIM 0999 #5
LD TR0
AND T0999
RSET bit_1s
; rung 9
LD=(300) A244 &1000
OUT TR0
AND bit_Ciclo
RSET bit_1s
LD TR0
ANDNOT bit_Ciclo
SET bit_1s
LD TR0
AND bit_1s
SET bit_Ciclo
LD TR0
ANDNOT bit_1s
RSET bit_Ciclo
; rung 10
LD P_On
MOV(021) #0 EmpyStr

### Section Maquina_01

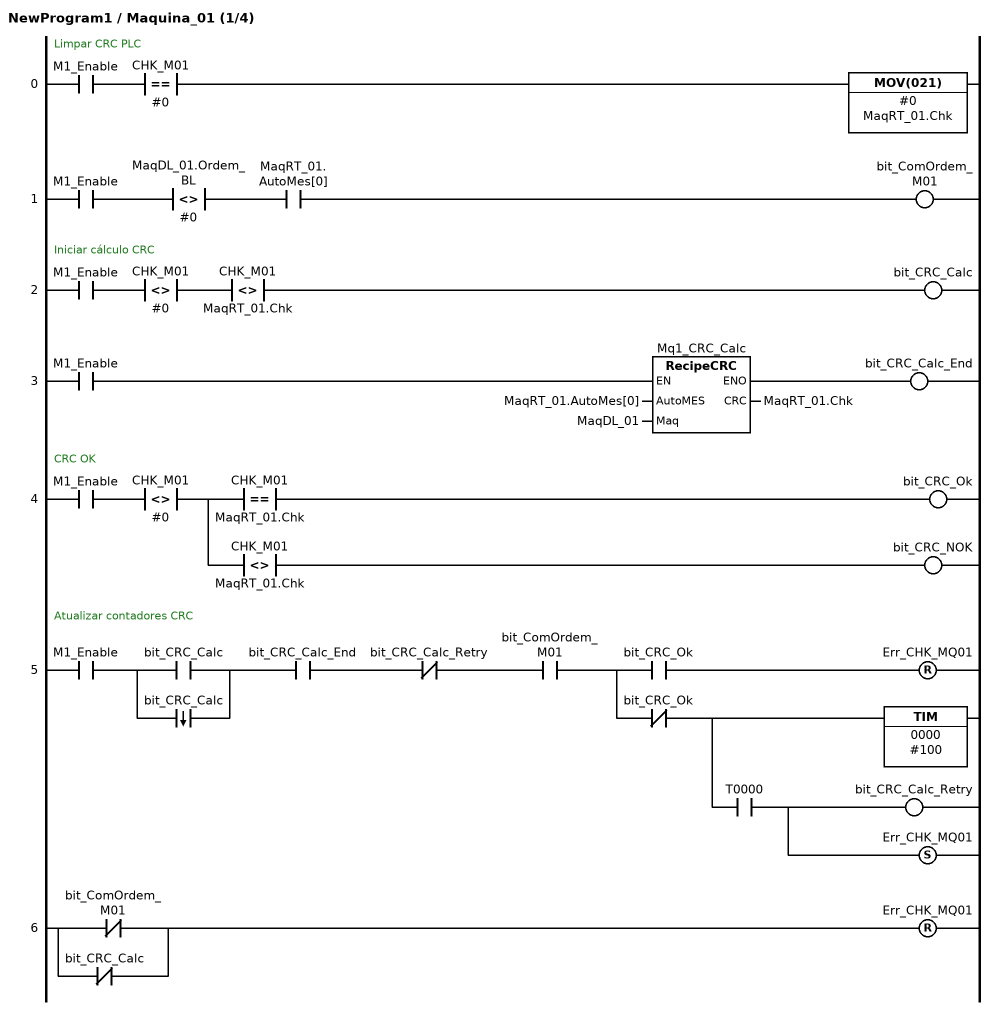
; rung 0: Limpar CRC PLC
LD M1_Enable
AND=(300) CHK_M01 #0
MOV(021) #0 MaqRT_01.Chk
; rung 1
LD M1_Enable
AND<>L(306) MaqDL_01.Ordem_BL #0
AND MaqRT_01.AutoMes[0]
OUT bit_ComOrdem_M01
; rung 2: Iniciar cálculo CRC
LD M1_Enable
AND<>(305) CHK_M01 #0
AND<>(305) CHK_M01 MaqRT_01.Chk
OUT bit_CRC_Calc
; rung 3
LD M1_Enable
CALL Mq1_CRC_Calc : RecipeCRC (AutoMES := MaqRT_01.AutoMes[0], Maq := MaqDL_01, CRC => MaqRT_01.Chk)
OUT bit_CRC_Calc_End
; rung 4: CRC OK
LD M1_Enable
AND<>(305) CHK_M01 #0
OUT TR0
AND=(300) CHK_M01 MaqRT_01.Chk
OUT bit_CRC_Ok
LD TR0
AND<>(305) CHK_M01 MaqRT_01.Chk
OUT bit_CRC_NOK
; rung 5: Atualizar contadores CRC
LD M1_Enable
LD bit_CRC_Calc
%OR bit_CRC_Calc
ANDLD
AND bit_CRC_Calc_End
ANDNOT bit_CRC_Calc_Retry
AND bit_ComOrdem_M01
OUT TR0
AND bit_CRC_Ok
RSET Err_CHK_MQ01
LD TR0
ANDNOT bit_CRC_Ok
TIM 0000 #100
AND T0000
OUT bit_CRC_Calc_Retry
SET Err_CHK_MQ01
; rung 6
LDNOT bit_ComOrdem_M01
ORNOT bit_CRC_Calc
RSET Err_CHK_MQ01

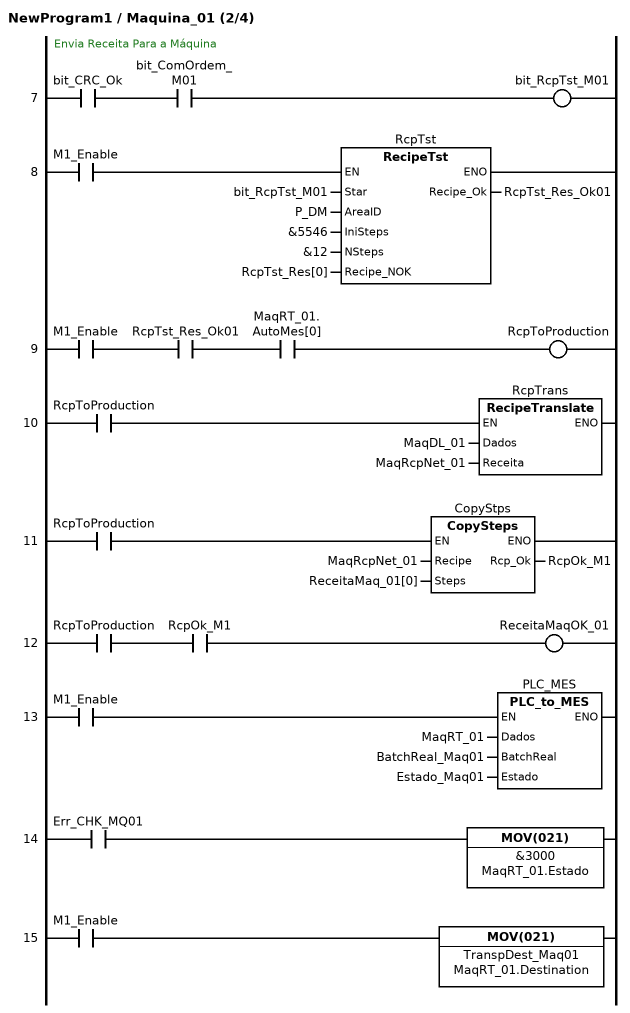
; rung 7: Envia Receita Para a Máquina
LD bit_CRC_Ok
AND bit_ComOrdem_M01
OUT bit_RcpTst_M01
; rung 8
LD M1_Enable
CALL RcpTst : RecipeTst (Star := bit_RcpTst_M01, AreaID := P_DM, IniSteps := &5546, NSteps := &12, Recipe_NOK := RcpTst_Res[0], Recipe_Ok => RcpTst_Res_Ok01)
; rung 9
LD M1_Enable
AND RcpTst_Res_Ok01
AND MaqRT_01.AutoMes[0]
OUT RcpToProduction
; rung 10
LD RcpToProduction
CALL RcpTrans : RecipeTranslate (Dados := MaqDL_01, Receita := MaqRcpNet_01)
; rung 11
LD RcpToProduction
CALL CopyStps : CopySteps (Recipe := MaqRcpNet_01, Steps := ReceitaMaq_01[0], Rcp_Ok => RcpOk_M1)
; rung 12
LD RcpToProduction
AND RcpOk_M1
OUT ReceitaMaqOK_01
; rung 13
LD M1_Enable
CALL PLC_MES : PLC_to_MES (Dados := MaqRT_01, BatchReal := BatchReal_Maq01, Estado := Estado_Maq01)
; rung 14
LD Err_CHK_MQ01
MOV(021) &3000 MaqRT_01.Estado
; rung 15
LD M1_Enable
MOV(021) TranspDest_Maq01 MaqRT_01.Destination

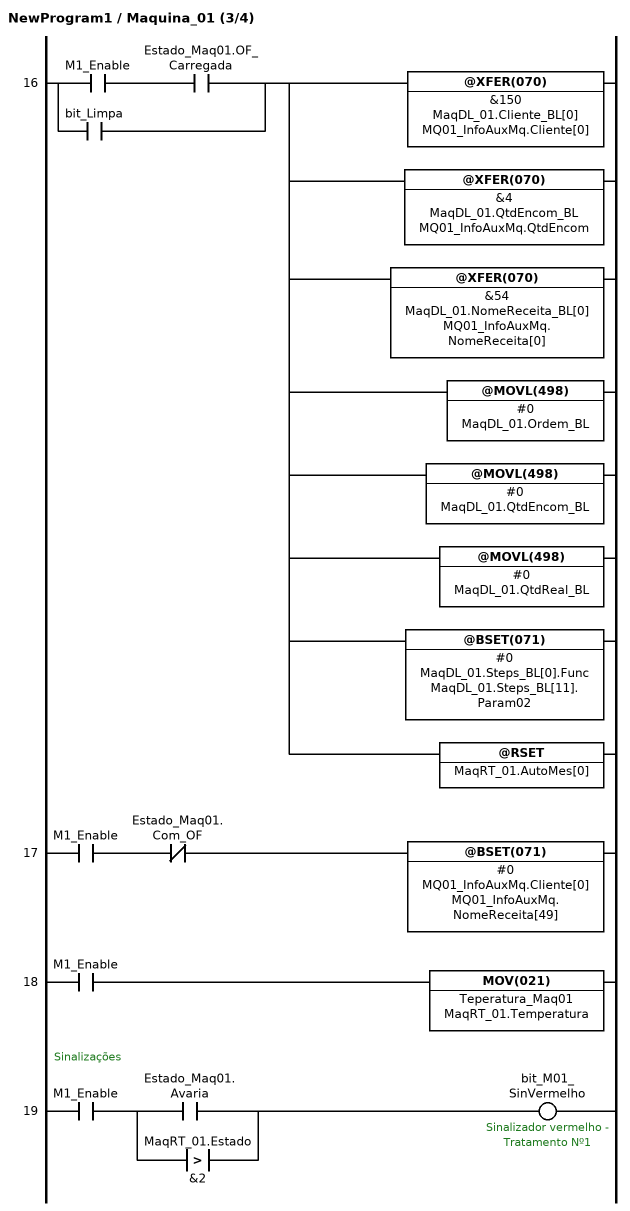
; rung 16
LD M1_Enable
AND Estado_Maq01.OF_Carregada
OR bit_Limpa
@XFER(070) &150 MaqDL_01.Cliente_BL[0] MQ01_InfoAuxMq.Cliente[0]
@XFER(070) &4 MaqDL_01.QtdEncom_BL MQ01_InfoAuxMq.QtdEncom
@XFER(070) &54 MaqDL_01.NomeReceita_BL[0] MQ01_InfoAuxMq.NomeReceita[0]
@MOVL(498) #0 MaqDL_01.Ordem_BL
@MOVL(498) #0 MaqDL_01.QtdEncom_BL
@MOVL(498) #0 MaqDL_01.QtdReal_BL
@BSET(071) #0 MaqDL_01.Steps_BL[0].Func MaqDL_01.Steps_BL[11].Param02
@RSET MaqRT_01.AutoMes[0]
; rung 17
LD M1_Enable
ANDNOT Estado_Maq01.Com_OF
@BSET(071) #0 MQ01_InfoAuxMq.Cliente[0] MQ01_InfoAuxMq.NomeReceita[49]
; rung 18
LD M1_Enable
MOV(021) Teperatura_Maq01 MaqRT_01.Temperatura
; rung 19: Sinalizações
LD M1_Enable
LD Estado_Maq01.Avaria
OR>(320) MaqRT_01.Estado &2
ANDLD
OUT bit_M01_SinVermelho  ; Sinalizador vermelho - Tratamento Nº1

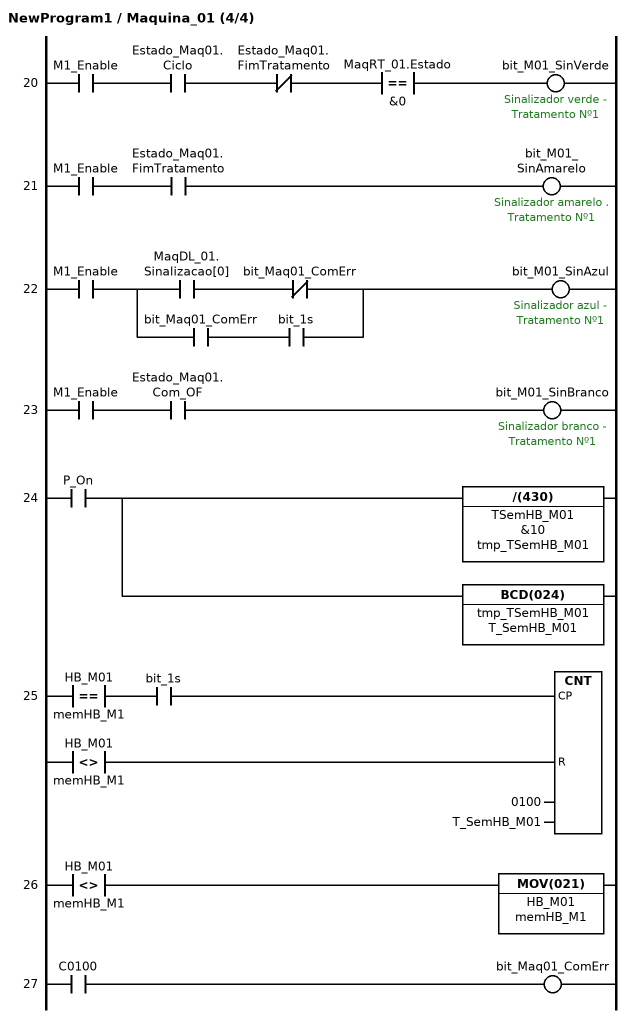
; rung 20
LD M1_Enable
AND Estado_Maq01.Ciclo
ANDNOT Estado_Maq01.FimTratamento
AND=(300) MaqRT_01.Estado &0
OUT bit_M01_SinVerde  ; Sinalizador verde - Tratamento Nº1
; rung 21
LD M1_Enable
AND Estado_Maq01.FimTratamento
OUT bit_M01_SinAmarelo  ; Sinalizador amarelo . Tratamento Nº1
; rung 22
LD M1_Enable
LD MaqDL_01.Sinalizacao[0]
ANDNOT bit_Maq01_ComErr
LD bit_Maq01_ComErr
AND bit_1s
ORLD
ANDLD
OUT bit_M01_SinAzul  ; Sinalizador azul - Tratamento Nº1
; rung 23
LD M1_Enable
AND Estado_Maq01.Com_OF
OUT bit_M01_SinBranco  ; Sinalizador branco - Tratamento Nº1
; rung 24
LD P_On
/(430) TSemHB_M01 &10 tmp_TSemHB_M01
BCD(024) tmp_TSemHB_M01 T_SemHB_M01
; rung 25
LD=(300) HB_M01 memHB_M1
AND bit_1s
LD<>(305) HB_M01 memHB_M1
CNT 0100 T_SemHB_M01
; rung 26
LD<>(305) HB_M01 memHB_M1
MOV(021) HB_M01 memHB_M1
; rung 27
LD C0100
OUT bit_Maq01_ComErr

### Section Maquina_02

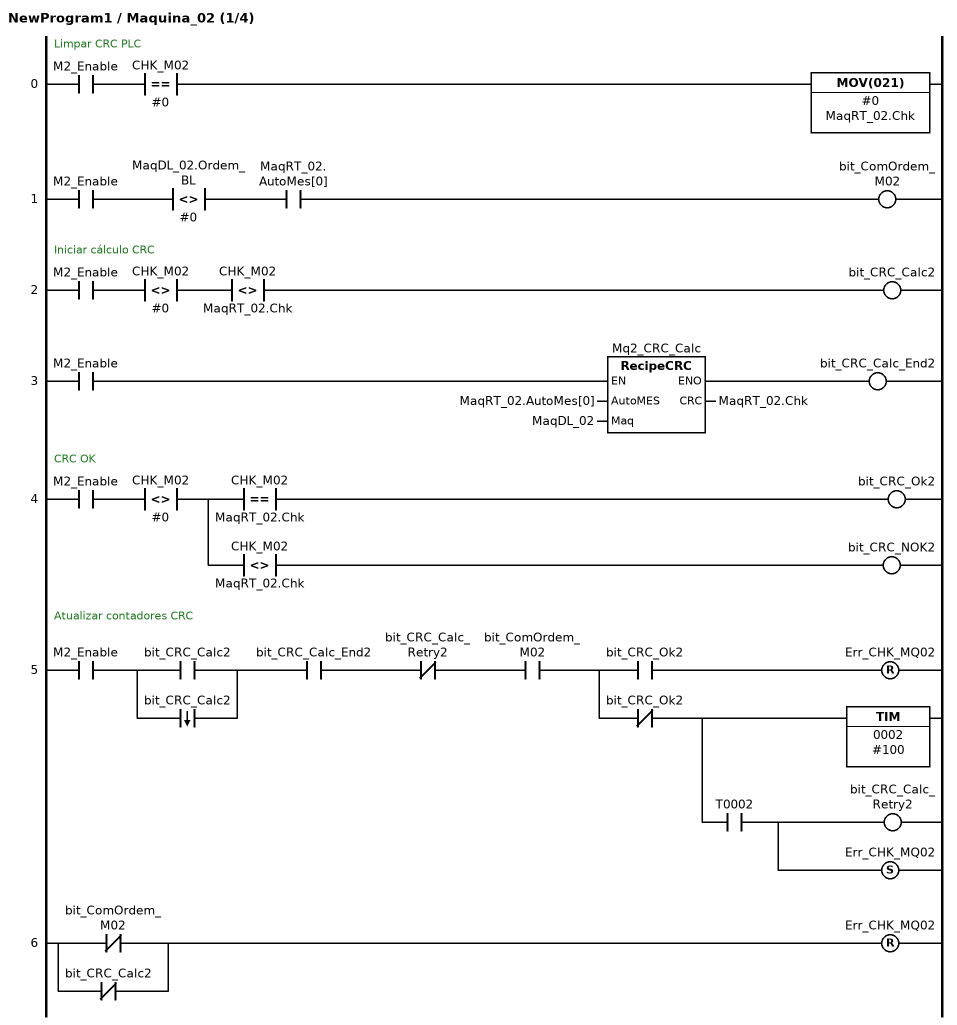
; rung 0: Limpar CRC PLC
LD M2_Enable
AND=(300) CHK_M02 #0
MOV(021) #0 MaqRT_02.Chk
; rung 1
LD M2_Enable
AND<>L(306) MaqDL_02.Ordem_BL #0
AND MaqRT_02.AutoMes[0]
OUT bit_ComOrdem_M02
; rung 2: Iniciar cálculo CRC
LD M2_Enable
AND<>(305) CHK_M02 #0
AND<>(305) CHK_M02 MaqRT_02.Chk
OUT bit_CRC_Calc2
; rung 3
LD M2_Enable
CALL Mq2_CRC_Calc : RecipeCRC (AutoMES := MaqRT_02.AutoMes[0], Maq := MaqDL_02, CRC => MaqRT_02.Chk)
OUT bit_CRC_Calc_End2
; rung 4: CRC OK
LD M2_Enable
AND<>(305) CHK_M02 #0
OUT TR0
AND=(300) CHK_M02 MaqRT_02.Chk
OUT bit_CRC_Ok2
LD TR0
AND<>(305) CHK_M02 MaqRT_02.Chk
OUT bit_CRC_NOK2
; rung 5: Atualizar contadores CRC
LD M2_Enable
LD bit_CRC_Calc2
%OR bit_CRC_Calc2
ANDLD
AND bit_CRC_Calc_End2
ANDNOT bit_CRC_Calc_Retry2
AND bit_ComOrdem_M02
OUT TR0
AND bit_CRC_Ok2
RSET Err_CHK_MQ02
LD TR0
ANDNOT bit_CRC_Ok2
TIM 0002 #100
AND T0002
OUT bit_CRC_Calc_Retry2
SET Err_CHK_MQ02
; rung 6
LDNOT bit_ComOrdem_M02
ORNOT bit_CRC_Calc2
RSET Err_CHK_MQ02

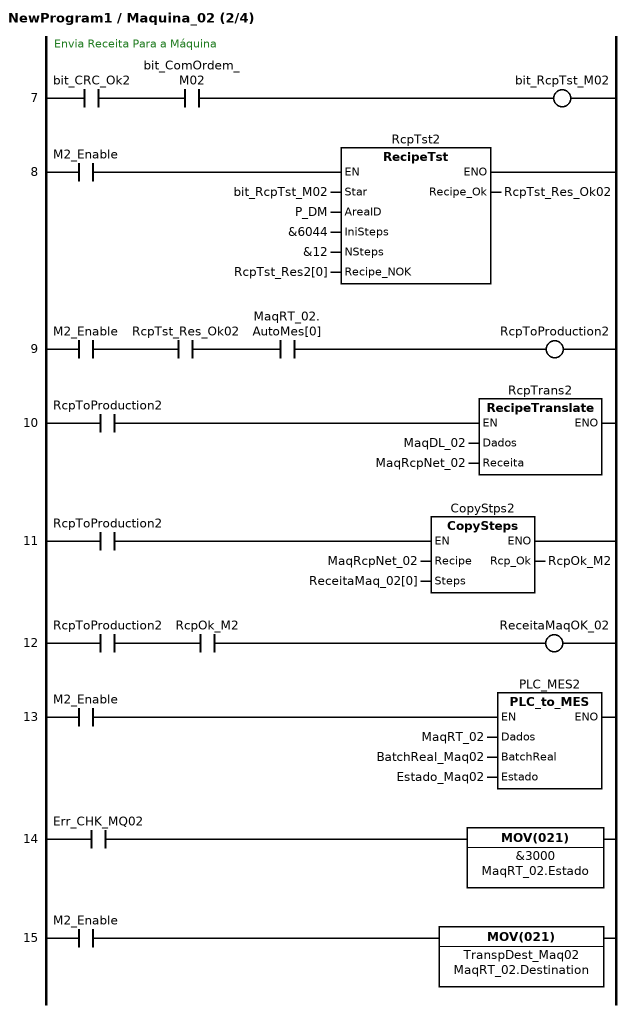
; rung 7: Envia Receita Para a Máquina
LD bit_CRC_Ok2
AND bit_ComOrdem_M02
OUT bit_RcpTst_M02
; rung 8
LD M2_Enable
CALL RcpTst2 : RecipeTst (Star := bit_RcpTst_M02, AreaID := P_DM, IniSteps := &6044, NSteps := &12, Recipe_NOK := RcpTst_Res2[0], Recipe_Ok => RcpTst_Res_Ok02)
; rung 9
LD M2_Enable
AND RcpTst_Res_Ok02
AND MaqRT_02.AutoMes[0]
OUT RcpToProduction2
; rung 10
LD RcpToProduction2
CALL RcpTrans2 : RecipeTranslate (Dados := MaqDL_02, Receita := MaqRcpNet_02)
; rung 11
LD RcpToProduction2
CALL CopyStps2 : CopySteps (Recipe := MaqRcpNet_02, Steps := ReceitaMaq_02[0], Rcp_Ok => RcpOk_M2)
; rung 12
LD RcpToProduction2
AND RcpOk_M2
OUT ReceitaMaqOK_02
; rung 13
LD M2_Enable
CALL PLC_MES2 : PLC_to_MES (Dados := MaqRT_02, BatchReal := BatchReal_Maq02, Estado := Estado_Maq02)
; rung 14
LD Err_CHK_MQ02
MOV(021) &3000 MaqRT_02.Estado
; rung 15
LD M2_Enable
MOV(021) TranspDest_Maq02 MaqRT_02.Destination

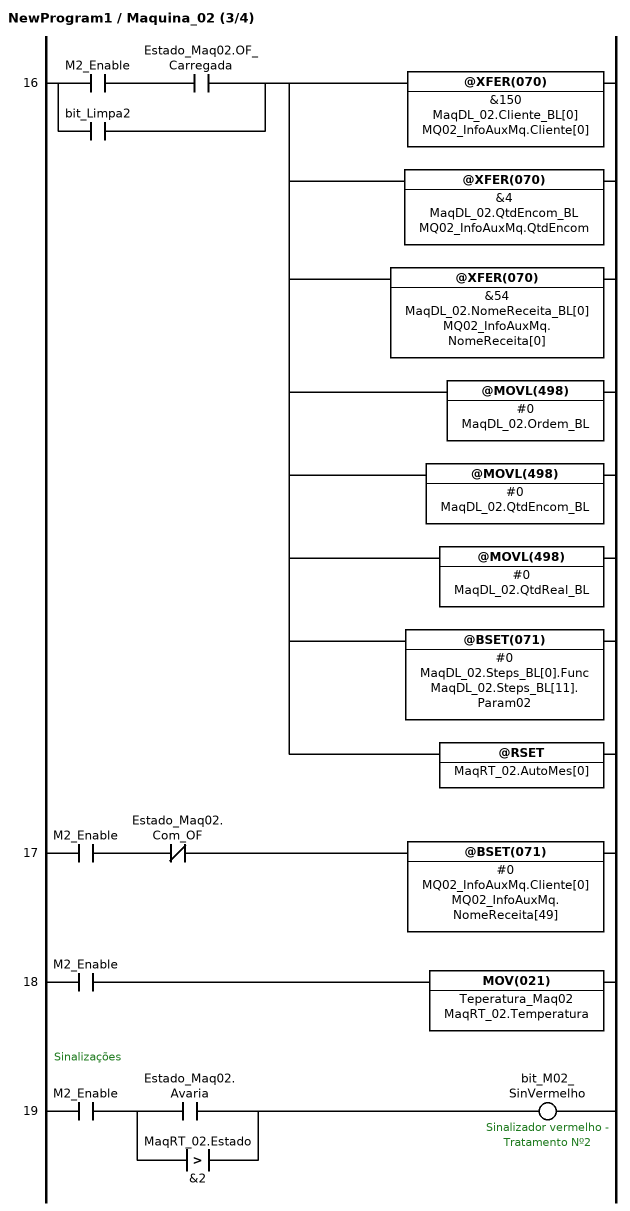
; rung 16
LD M2_Enable
AND Estado_Maq02.OF_Carregada
OR bit_Limpa2
@XFER(070) &150 MaqDL_02.Cliente_BL[0] MQ02_InfoAuxMq.Cliente[0]
@XFER(070) &4 MaqDL_02.QtdEncom_BL MQ02_InfoAuxMq.QtdEncom
@XFER(070) &54 MaqDL_02.NomeReceita_BL[0] MQ02_InfoAuxMq.NomeReceita[0]
@MOVL(498) #0 MaqDL_02.Ordem_BL
@MOVL(498) #0 MaqDL_02.QtdEncom_BL
@MOVL(498) #0 MaqDL_02.QtdReal_BL
@BSET(071) #0 MaqDL_02.Steps_BL[0].Func MaqDL_02.Steps_BL[11].Param02
@RSET MaqRT_02.AutoMes[0]
; rung 17
LD M2_Enable
ANDNOT Estado_Maq02.Com_OF
@BSET(071) #0 MQ02_InfoAuxMq.Cliente[0] MQ02_InfoAuxMq.NomeReceita[49]
; rung 18
LD M2_Enable
MOV(021) Teperatura_Maq02 MaqRT_02.Temperatura
; rung 19: Sinalizações
LD M2_Enable
LD Estado_Maq02.Avaria
OR>(320) MaqRT_02.Estado &2
ANDLD
OUT bit_M02_SinVermelho  ; Sinalizador vermelho - Tratamento Nº2

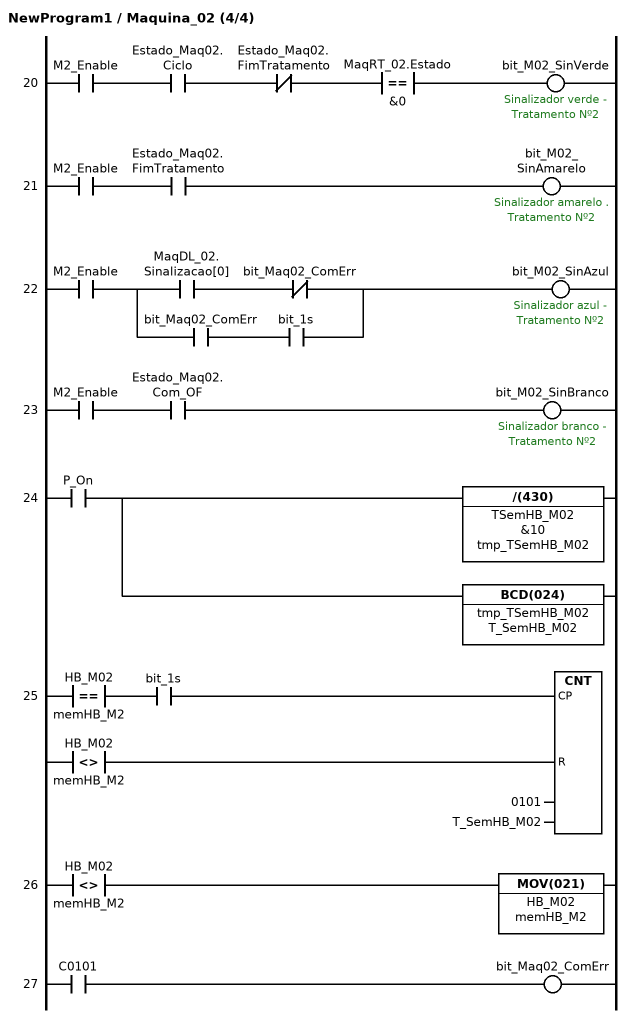
; rung 20
LD M2_Enable
AND Estado_Maq02.Ciclo
ANDNOT Estado_Maq02.FimTratamento
AND=(300) MaqRT_02.Estado &0
OUT bit_M02_SinVerde  ; Sinalizador verde - Tratamento Nº2
; rung 21
LD M2_Enable
AND Estado_Maq02.FimTratamento
OUT bit_M02_SinAmarelo  ; Sinalizador amarelo . Tratamento Nº2
; rung 22
LD M2_Enable
LD MaqDL_02.Sinalizacao[0]
ANDNOT bit_Maq02_ComErr
LD bit_Maq02_ComErr
AND bit_1s
ORLD
ANDLD
OUT bit_M02_SinAzul  ; Sinalizador azul - Tratamento Nº2
; rung 23
LD M2_Enable
AND Estado_Maq02.Com_OF
OUT bit_M02_SinBranco  ; Sinalizador branco - Tratamento Nº2
; rung 24
LD P_On
/(430) TSemHB_M02 &10 tmp_TSemHB_M02
BCD(024) tmp_TSemHB_M02 T_SemHB_M02
; rung 25
LD=(300) HB_M02 memHB_M2
AND bit_1s
LD<>(305) HB_M02 memHB_M2
CNT 0101 T_SemHB_M02
; rung 26
LD<>(305) HB_M02 memHB_M2
MOV(021) HB_M02 memHB_M2
; rung 27
LD C0101
OUT bit_Maq02_ComErr

### Section Maquina_03

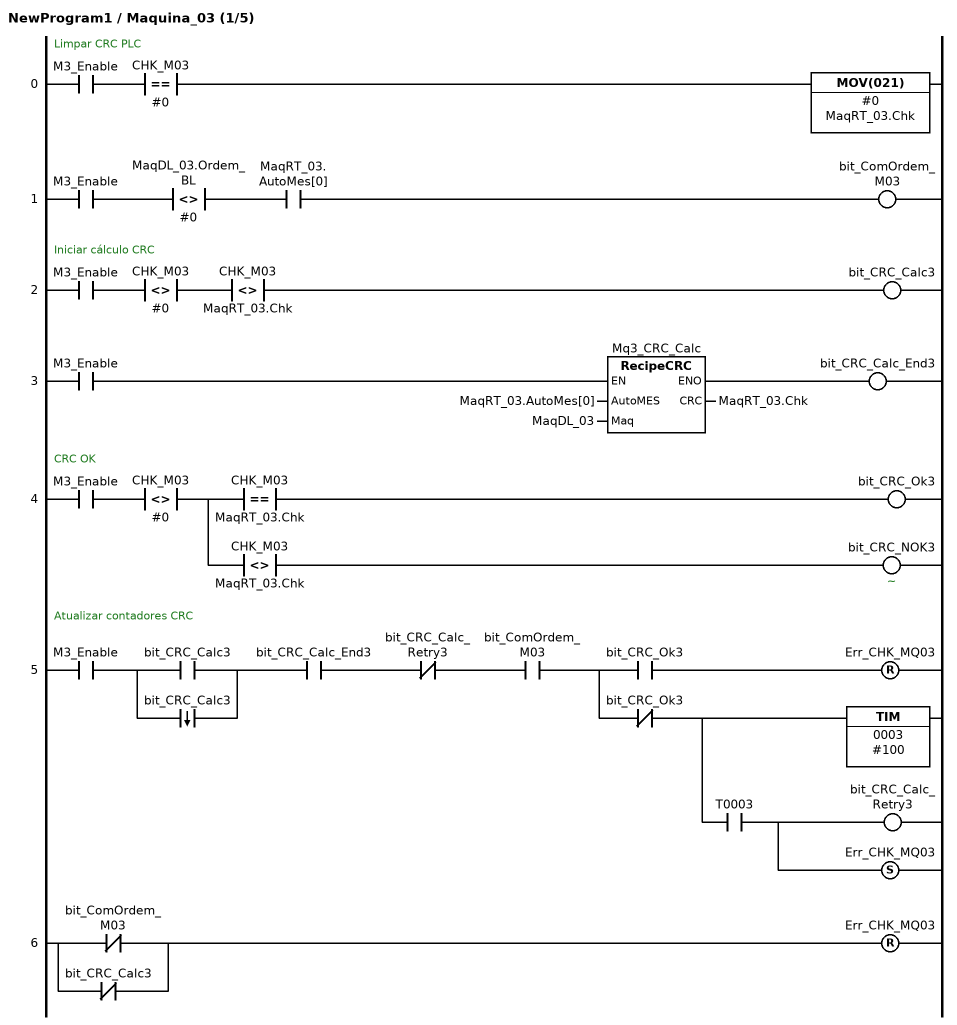
; rung 0: Limpar CRC PLC
LD M3_Enable
AND=(300) CHK_M03 #0
MOV(021) #0 MaqRT_03.Chk
; rung 1
LD M3_Enable
AND<>L(306) MaqDL_03.Ordem_BL #0
AND MaqRT_03.AutoMes[0]
OUT bit_ComOrdem_M03
; rung 2: Iniciar cálculo CRC
LD M3_Enable
AND<>(305) CHK_M03 #0
AND<>(305) CHK_M03 MaqRT_03.Chk
OUT bit_CRC_Calc3
; rung 3
LD M3_Enable
CALL Mq3_CRC_Calc : RecipeCRC (AutoMES := MaqRT_03.AutoMes[0], Maq := MaqDL_03, CRC => MaqRT_03.Chk)
OUT bit_CRC_Calc_End3
; rung 4: CRC OK
LD M3_Enable
AND<>(305) CHK_M03 #0
OUT TR0
AND=(300) CHK_M03 MaqRT_03.Chk
OUT bit_CRC_Ok3
LD TR0
AND<>(305) CHK_M03 MaqRT_03.Chk
OUT bit_CRC_NOK3  ; ~
; rung 5: Atualizar contadores CRC
LD M3_Enable
LD bit_CRC_Calc3
%OR bit_CRC_Calc3
ANDLD
AND bit_CRC_Calc_End3
ANDNOT bit_CRC_Calc_Retry3
AND bit_ComOrdem_M03
OUT TR0
AND bit_CRC_Ok3
RSET Err_CHK_MQ03
LD TR0
ANDNOT bit_CRC_Ok3
TIM 0003 #100
AND T0003
OUT bit_CRC_Calc_Retry3
SET Err_CHK_MQ03
; rung 6
LDNOT bit_ComOrdem_M03
ORNOT bit_CRC_Calc3
RSET Err_CHK_MQ03

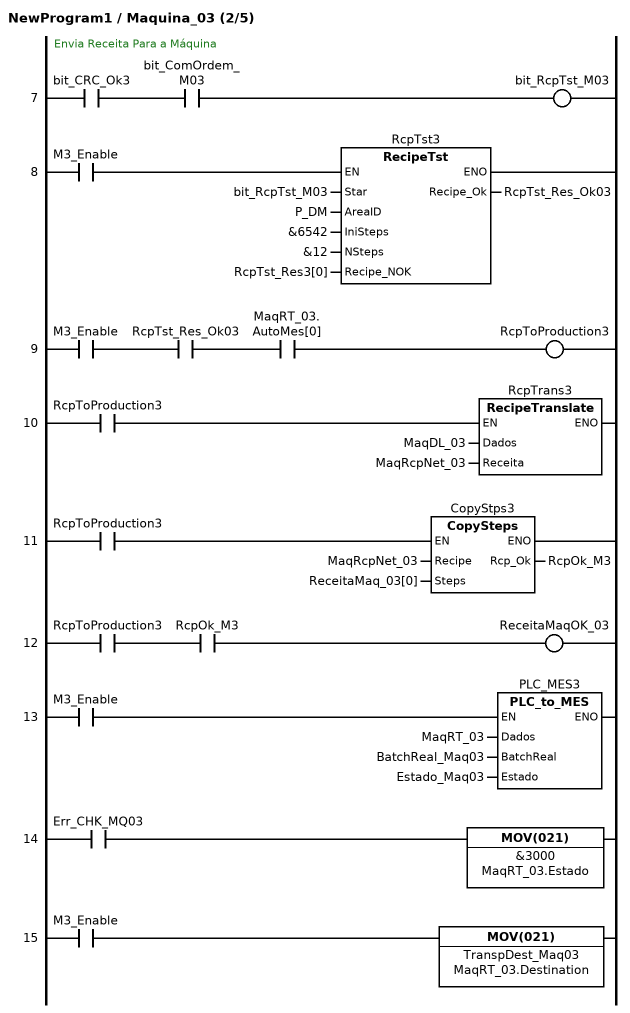
; rung 7: Envia Receita Para a Máquina
LD bit_CRC_Ok3
AND bit_ComOrdem_M03
OUT bit_RcpTst_M03
; rung 8
LD M3_Enable
CALL RcpTst3 : RecipeTst (Star := bit_RcpTst_M03, AreaID := P_DM, IniSteps := &6542, NSteps := &12, Recipe_NOK := RcpTst_Res3[0], Recipe_Ok => RcpTst_Res_Ok03)
; rung 9
LD M3_Enable
AND RcpTst_Res_Ok03
AND MaqRT_03.AutoMes[0]
OUT RcpToProduction3
; rung 10
LD RcpToProduction3
CALL RcpTrans3 : RecipeTranslate (Dados := MaqDL_03, Receita := MaqRcpNet_03)
; rung 11
LD RcpToProduction3
CALL CopyStps3 : CopySteps (Recipe := MaqRcpNet_03, Steps := ReceitaMaq_03[0], Rcp_Ok => RcpOk_M3)
; rung 12
LD RcpToProduction3
AND RcpOk_M3
OUT ReceitaMaqOK_03
; rung 13
LD M3_Enable
CALL PLC_MES3 : PLC_to_MES (Dados := MaqRT_03, BatchReal := BatchReal_Maq03, Estado := Estado_Maq03)
; rung 14
LD Err_CHK_MQ03
MOV(021) &3000 MaqRT_03.Estado
; rung 15
LD M3_Enable
MOV(021) TranspDest_Maq03 MaqRT_03.Destination

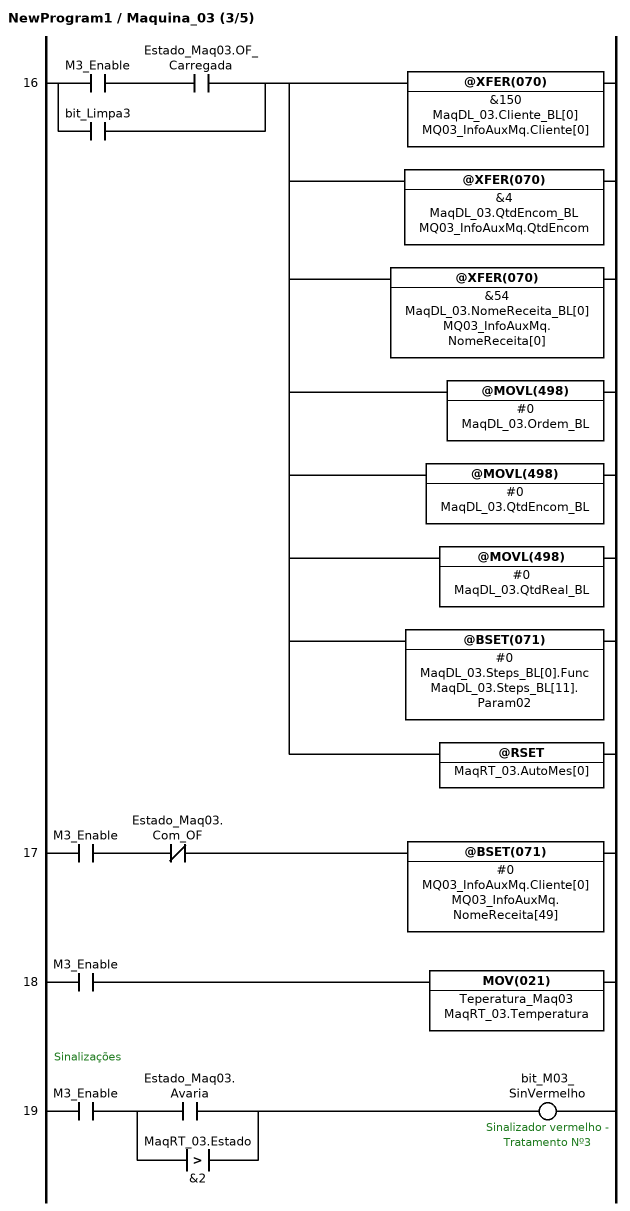
; rung 16
LD M3_Enable
AND Estado_Maq03.OF_Carregada
OR bit_Limpa3
@XFER(070) &150 MaqDL_03.Cliente_BL[0] MQ03_InfoAuxMq.Cliente[0]
@XFER(070) &4 MaqDL_03.QtdEncom_BL MQ03_InfoAuxMq.QtdEncom
@XFER(070) &54 MaqDL_03.NomeReceita_BL[0] MQ03_InfoAuxMq.NomeReceita[0]
@MOVL(498) #0 MaqDL_03.Ordem_BL
@MOVL(498) #0 MaqDL_03.QtdEncom_BL
@MOVL(498) #0 MaqDL_03.QtdReal_BL
@BSET(071) #0 MaqDL_03.Steps_BL[0].Func MaqDL_03.Steps_BL[11].Param02
@RSET MaqRT_03.AutoMes[0]
; rung 17
LD M3_Enable
ANDNOT Estado_Maq03.Com_OF
@BSET(071) #0 MQ03_InfoAuxMq.Cliente[0] MQ03_InfoAuxMq.NomeReceita[49]
; rung 18
LD M3_Enable
MOV(021) Teperatura_Maq03 MaqRT_03.Temperatura
; rung 19: Sinalizações
LD M3_Enable
LD Estado_Maq03.Avaria
OR>(320) MaqRT_03.Estado &2
ANDLD
OUT bit_M03_SinVermelho  ; Sinalizador vermelho - Tratamento Nº3

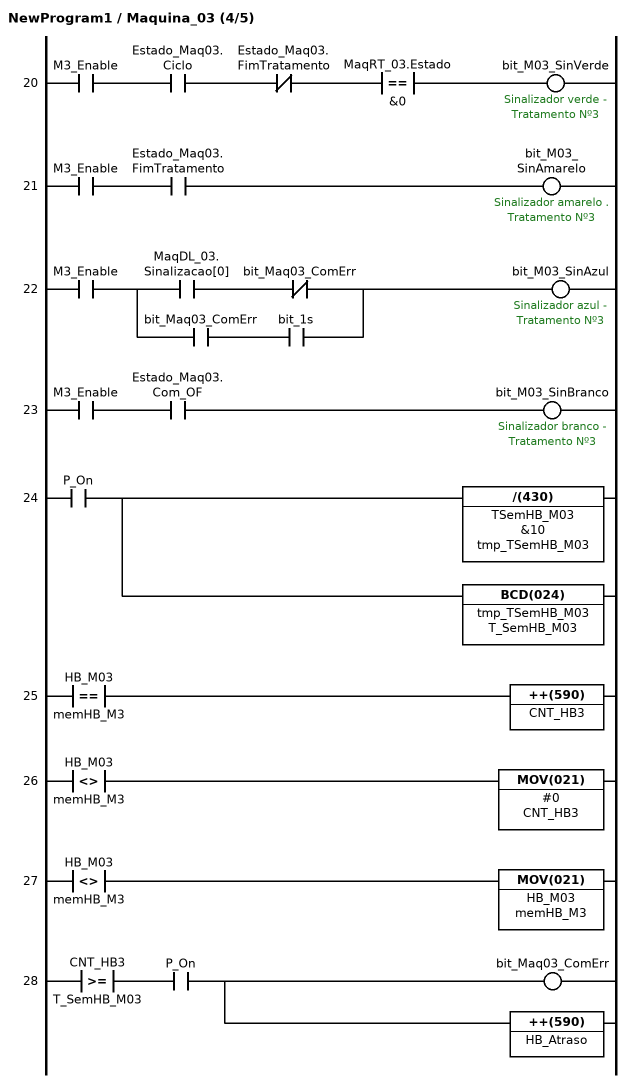
; rung 20
LD M3_Enable
AND Estado_Maq03.Ciclo
ANDNOT Estado_Maq03.FimTratamento
AND=(300) MaqRT_03.Estado &0
OUT bit_M03_SinVerde  ; Sinalizador verde - Tratamento Nº3
; rung 21
LD M3_Enable
AND Estado_Maq03.FimTratamento
OUT bit_M03_SinAmarelo  ; Sinalizador amarelo . Tratamento Nº3
; rung 22
LD M3_Enable
LD MaqDL_03.Sinalizacao[0]
ANDNOT bit_Maq03_ComErr
LD bit_Maq03_ComErr
AND bit_1s
ORLD
ANDLD
OUT bit_M03_SinAzul  ; Sinalizador azul - Tratamento Nº3
; rung 23
LD M3_Enable
AND Estado_Maq03.Com_OF
OUT bit_M03_SinBranco  ; Sinalizador branco - Tratamento Nº3
; rung 24
LD P_On
/(430) TSemHB_M03 &10 tmp_TSemHB_M03
BCD(024) tmp_TSemHB_M03 T_SemHB_M03
; rung 25
LD=(300) HB_M03 memHB_M3
++(590) CNT_HB3
; rung 26
LD<>(305) HB_M03 memHB_M3
MOV(021) #0 CNT_HB3
; rung 27
LD<>(305) HB_M03 memHB_M3
MOV(021) HB_M03 memHB_M3
; rung 28
LD>=(325) CNT_HB3 T_SemHB_M03
AND P_On
OUT bit_Maq03_ComErr
++(590) HB_Atraso

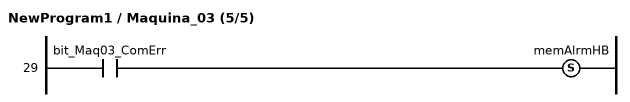
; rung 29
LD bit_Maq03_ComErr
SET memAlrmHB

### Section Maquina_04

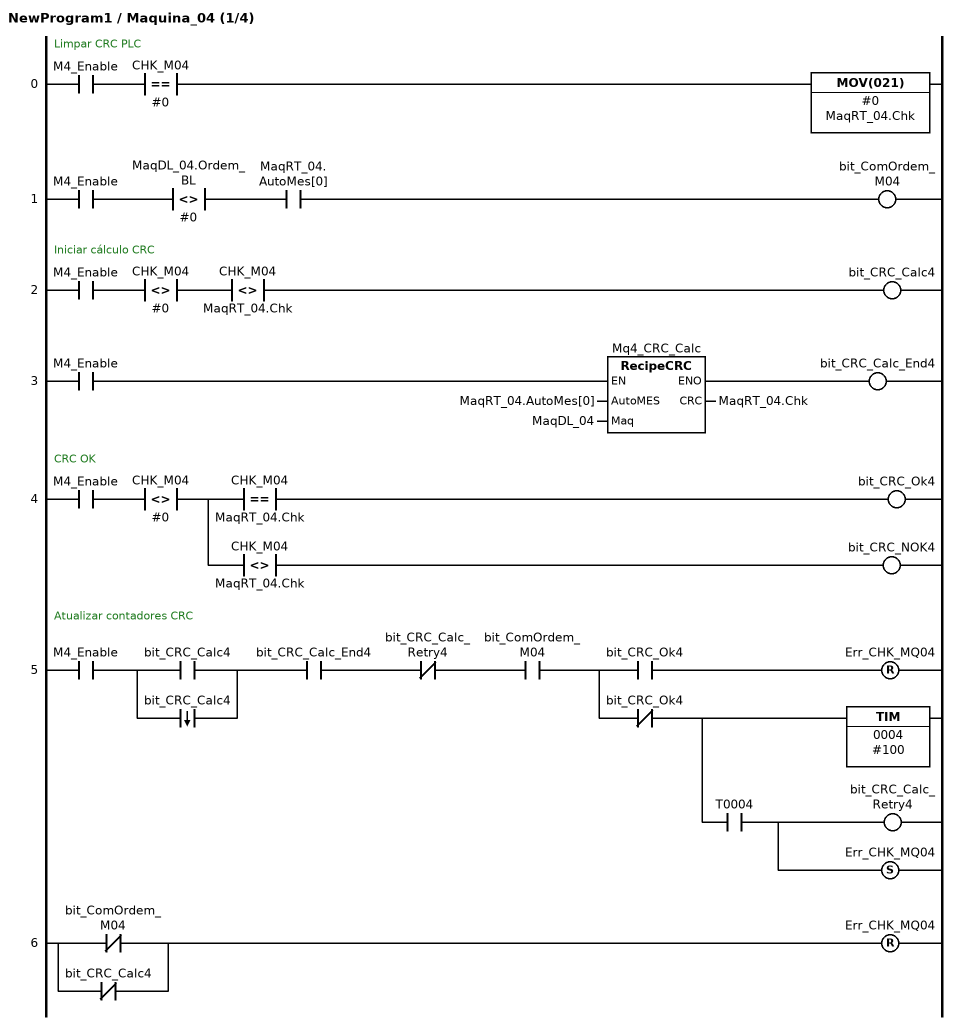
; rung 0: Limpar CRC PLC
LD M4_Enable
AND=(300) CHK_M04 #0
MOV(021) #0 MaqRT_04.Chk
; rung 1
LD M4_Enable
AND<>L(306) MaqDL_04.Ordem_BL #0
AND MaqRT_04.AutoMes[0]
OUT bit_ComOrdem_M04
; rung 2: Iniciar cálculo CRC
LD M4_Enable
AND<>(305) CHK_M04 #0
AND<>(305) CHK_M04 MaqRT_04.Chk
OUT bit_CRC_Calc4
; rung 3
LD M4_Enable
CALL Mq4_CRC_Calc : RecipeCRC (AutoMES := MaqRT_04.AutoMes[0], Maq := MaqDL_04, CRC => MaqRT_04.Chk)
OUT bit_CRC_Calc_End4
; rung 4: CRC OK
LD M4_Enable
AND<>(305) CHK_M04 #0
OUT TR0
AND=(300) CHK_M04 MaqRT_04.Chk
OUT bit_CRC_Ok4
LD TR0
AND<>(305) CHK_M04 MaqRT_04.Chk
OUT bit_CRC_NOK4
; rung 5: Atualizar contadores CRC
LD M4_Enable
LD bit_CRC_Calc4
%OR bit_CRC_Calc4
ANDLD
AND bit_CRC_Calc_End4
ANDNOT bit_CRC_Calc_Retry4
AND bit_ComOrdem_M04
OUT TR0
AND bit_CRC_Ok4
RSET Err_CHK_MQ04
LD TR0
ANDNOT bit_CRC_Ok4
TIM 0004 #100
AND T0004
OUT bit_CRC_Calc_Retry4
SET Err_CHK_MQ04
; rung 6
LDNOT bit_ComOrdem_M04
ORNOT bit_CRC_Calc4
RSET Err_CHK_MQ04

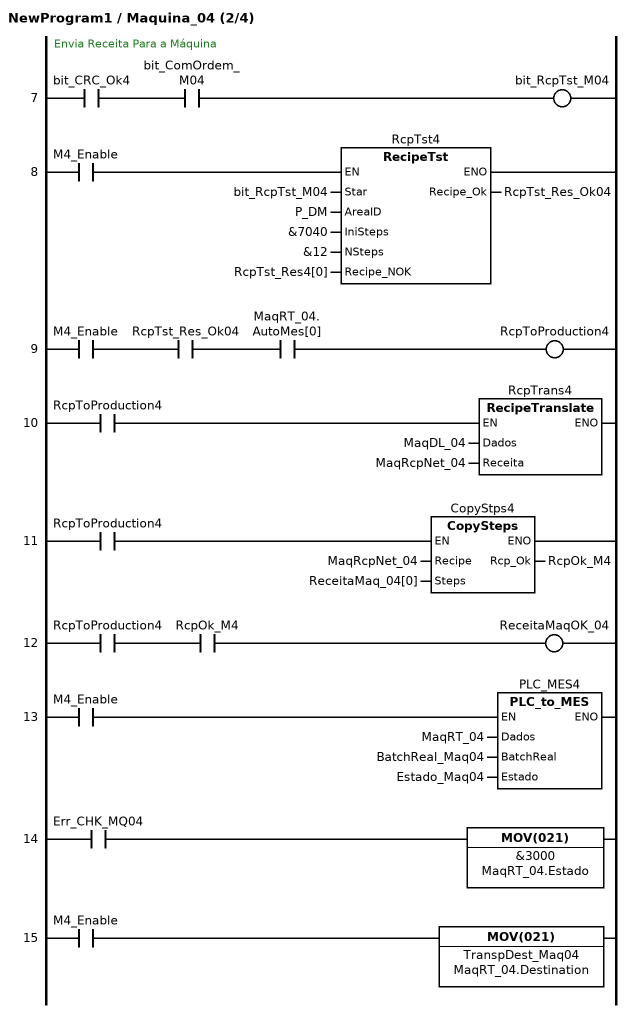
; rung 7: Envia Receita Para a Máquina
LD bit_CRC_Ok4
AND bit_ComOrdem_M04
OUT bit_RcpTst_M04
; rung 8
LD M4_Enable
CALL RcpTst4 : RecipeTst (Star := bit_RcpTst_M04, AreaID := P_DM, IniSteps := &7040, NSteps := &12, Recipe_NOK := RcpTst_Res4[0], Recipe_Ok => RcpTst_Res_Ok04)
; rung 9
LD M4_Enable
AND RcpTst_Res_Ok04
AND MaqRT_04.AutoMes[0]
OUT RcpToProduction4
; rung 10
LD RcpToProduction4
CALL RcpTrans4 : RecipeTranslate (Dados := MaqDL_04, Receita := MaqRcpNet_04)
; rung 11
LD RcpToProduction4
CALL CopyStps4 : CopySteps (Recipe := MaqRcpNet_04, Steps := ReceitaMaq_04[0], Rcp_Ok => RcpOk_M4)
; rung 12
LD RcpToProduction4
AND RcpOk_M4
OUT ReceitaMaqOK_04
; rung 13
LD M4_Enable
CALL PLC_MES4 : PLC_to_MES (Dados := MaqRT_04, BatchReal := BatchReal_Maq04, Estado := Estado_Maq04)
; rung 14
LD Err_CHK_MQ04
MOV(021) &3000 MaqRT_04.Estado
; rung 15
LD M4_Enable
MOV(021) TranspDest_Maq04 MaqRT_04.Destination

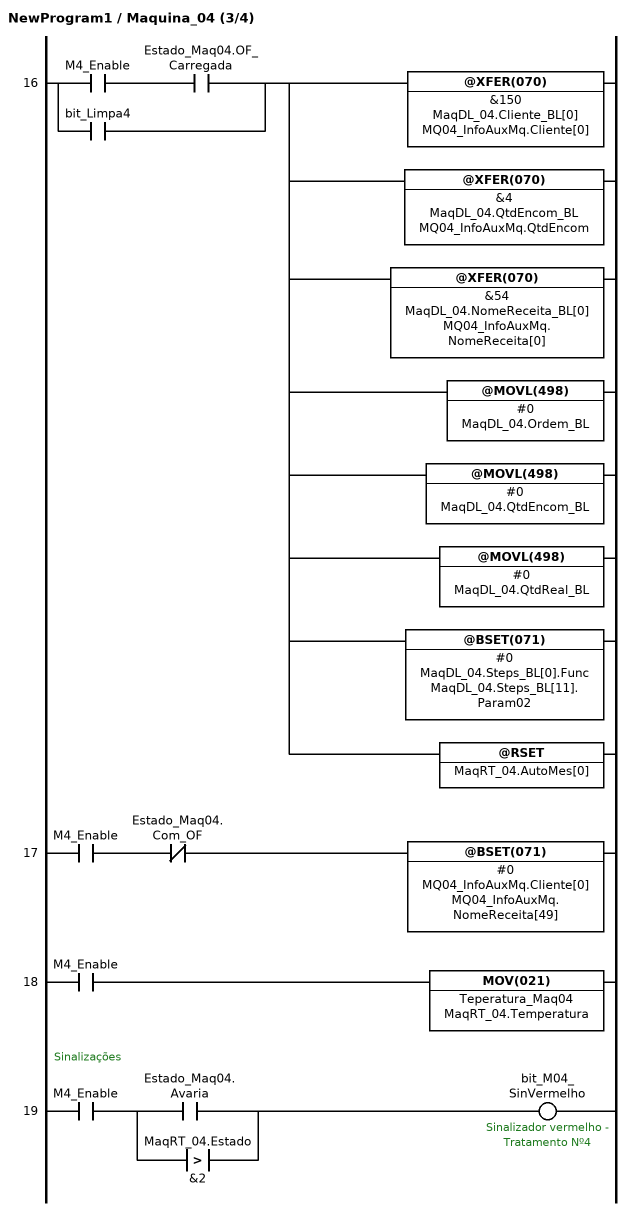
; rung 16
LD M4_Enable
AND Estado_Maq04.OF_Carregada
OR bit_Limpa4
@XFER(070) &150 MaqDL_04.Cliente_BL[0] MQ04_InfoAuxMq.Cliente[0]
@XFER(070) &4 MaqDL_04.QtdEncom_BL MQ04_InfoAuxMq.QtdEncom
@XFER(070) &54 MaqDL_04.NomeReceita_BL[0] MQ04_InfoAuxMq.NomeReceita[0]
@MOVL(498) #0 MaqDL_04.Ordem_BL
@MOVL(498) #0 MaqDL_04.QtdEncom_BL
@MOVL(498) #0 MaqDL_04.QtdReal_BL
@BSET(071) #0 MaqDL_04.Steps_BL[0].Func MaqDL_04.Steps_BL[11].Param02
@RSET MaqRT_04.AutoMes[0]
; rung 17
LD M4_Enable
ANDNOT Estado_Maq04.Com_OF
@BSET(071) #0 MQ04_InfoAuxMq.Cliente[0] MQ04_InfoAuxMq.NomeReceita[49]
; rung 18
LD M4_Enable
MOV(021) Teperatura_Maq04 MaqRT_04.Temperatura
; rung 19: Sinalizações
LD M4_Enable
LD Estado_Maq04.Avaria
OR>(320) MaqRT_04.Estado &2
ANDLD
OUT bit_M04_SinVermelho  ; Sinalizador vermelho - Tratamento Nº4

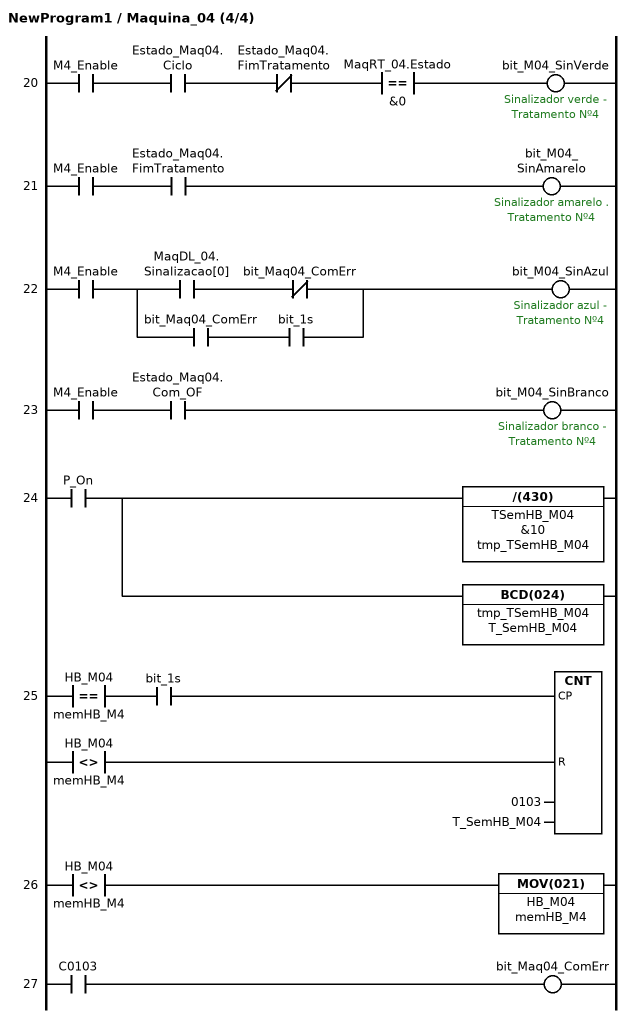
; rung 20
LD M4_Enable
AND Estado_Maq04.Ciclo
ANDNOT Estado_Maq04.FimTratamento
AND=(300) MaqRT_04.Estado &0
OUT bit_M04_SinVerde  ; Sinalizador verde - Tratamento Nº4
; rung 21
LD M4_Enable
AND Estado_Maq04.FimTratamento
OUT bit_M04_SinAmarelo  ; Sinalizador amarelo . Tratamento Nº4
; rung 22
LD M4_Enable
LD MaqDL_04.Sinalizacao[0]
ANDNOT bit_Maq04_ComErr
LD bit_Maq04_ComErr
AND bit_1s
ORLD
ANDLD
OUT bit_M04_SinAzul  ; Sinalizador azul - Tratamento Nº4
; rung 23
LD M4_Enable
AND Estado_Maq04.Com_OF
OUT bit_M04_SinBranco  ; Sinalizador branco - Tratamento Nº4
; rung 24
LD P_On
/(430) TSemHB_M04 &10 tmp_TSemHB_M04
BCD(024) tmp_TSemHB_M04 T_SemHB_M04
; rung 25
LD=(300) HB_M04 memHB_M4
AND bit_1s
LD<>(305) HB_M04 memHB_M4
CNT 0103 T_SemHB_M04
; rung 26
LD<>(305) HB_M04 memHB_M4
MOV(021) HB_M04 memHB_M4
; rung 27
LD C0103
OUT bit_Maq04_ComErr

### Section Maquina_05

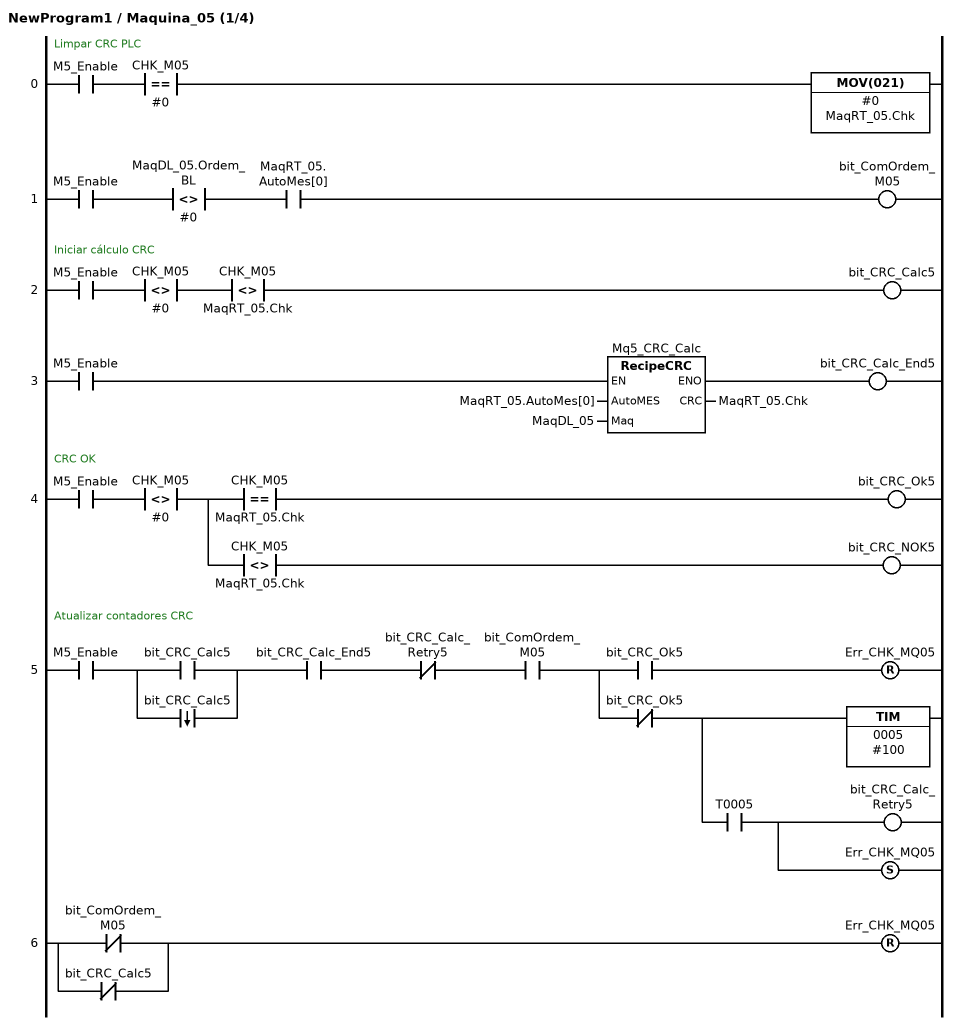
; rung 0: Limpar CRC PLC
LD M5_Enable
AND=(300) CHK_M05 #0
MOV(021) #0 MaqRT_05.Chk
; rung 1
LD M5_Enable
AND<>L(306) MaqDL_05.Ordem_BL #0
AND MaqRT_05.AutoMes[0]
OUT bit_ComOrdem_M05
; rung 2: Iniciar cálculo CRC
LD M5_Enable
AND<>(305) CHK_M05 #0
AND<>(305) CHK_M05 MaqRT_05.Chk
OUT bit_CRC_Calc5
; rung 3
LD M5_Enable
CALL Mq5_CRC_Calc : RecipeCRC (AutoMES := MaqRT_05.AutoMes[0], Maq := MaqDL_05, CRC => MaqRT_05.Chk)
OUT bit_CRC_Calc_End5
; rung 4: CRC OK
LD M5_Enable
AND<>(305) CHK_M05 #0
OUT TR0
AND=(300) CHK_M05 MaqRT_05.Chk
OUT bit_CRC_Ok5
LD TR0
AND<>(305) CHK_M05 MaqRT_05.Chk
OUT bit_CRC_NOK5
; rung 5: Atualizar contadores CRC
LD M5_Enable
LD bit_CRC_Calc5
%OR bit_CRC_Calc5
ANDLD
AND bit_CRC_Calc_End5
ANDNOT bit_CRC_Calc_Retry5
AND bit_ComOrdem_M05
OUT TR0
AND bit_CRC_Ok5
RSET Err_CHK_MQ05
LD TR0
ANDNOT bit_CRC_Ok5
TIM 0005 #100
AND T0005
OUT bit_CRC_Calc_Retry5
SET Err_CHK_MQ05
; rung 6
LDNOT bit_ComOrdem_M05
ORNOT bit_CRC_Calc5
RSET Err_CHK_MQ05

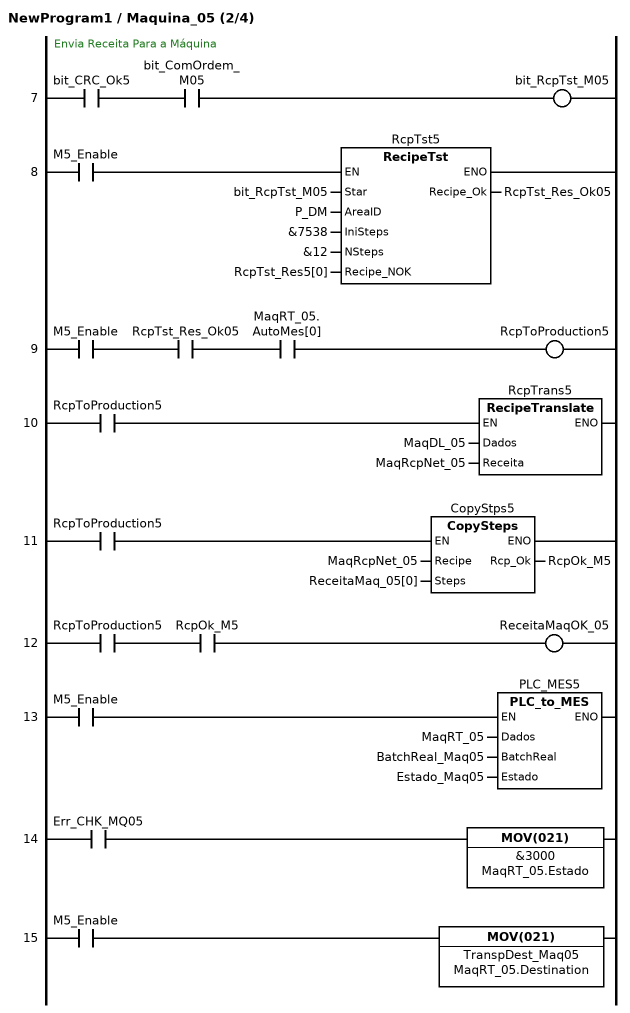
; rung 7: Envia Receita Para a Máquina
LD bit_CRC_Ok5
AND bit_ComOrdem_M05
OUT bit_RcpTst_M05
; rung 8
LD M5_Enable
CALL RcpTst5 : RecipeTst (Star := bit_RcpTst_M05, AreaID := P_DM, IniSteps := &7538, NSteps := &12, Recipe_NOK := RcpTst_Res5[0], Recipe_Ok => RcpTst_Res_Ok05)
; rung 9
LD M5_Enable
AND RcpTst_Res_Ok05
AND MaqRT_05.AutoMes[0]
OUT RcpToProduction5
; rung 10
LD RcpToProduction5
CALL RcpTrans5 : RecipeTranslate (Dados := MaqDL_05, Receita := MaqRcpNet_05)
; rung 11
LD RcpToProduction5
CALL CopyStps5 : CopySteps (Recipe := MaqRcpNet_05, Steps := ReceitaMaq_05[0], Rcp_Ok => RcpOk_M5)
; rung 12
LD RcpToProduction5
AND RcpOk_M5
OUT ReceitaMaqOK_05
; rung 13
LD M5_Enable
CALL PLC_MES5 : PLC_to_MES (Dados := MaqRT_05, BatchReal := BatchReal_Maq05, Estado := Estado_Maq05)
; rung 14
LD Err_CHK_MQ05
MOV(021) &3000 MaqRT_05.Estado
; rung 15
LD M5_Enable
MOV(021) TranspDest_Maq05 MaqRT_05.Destination

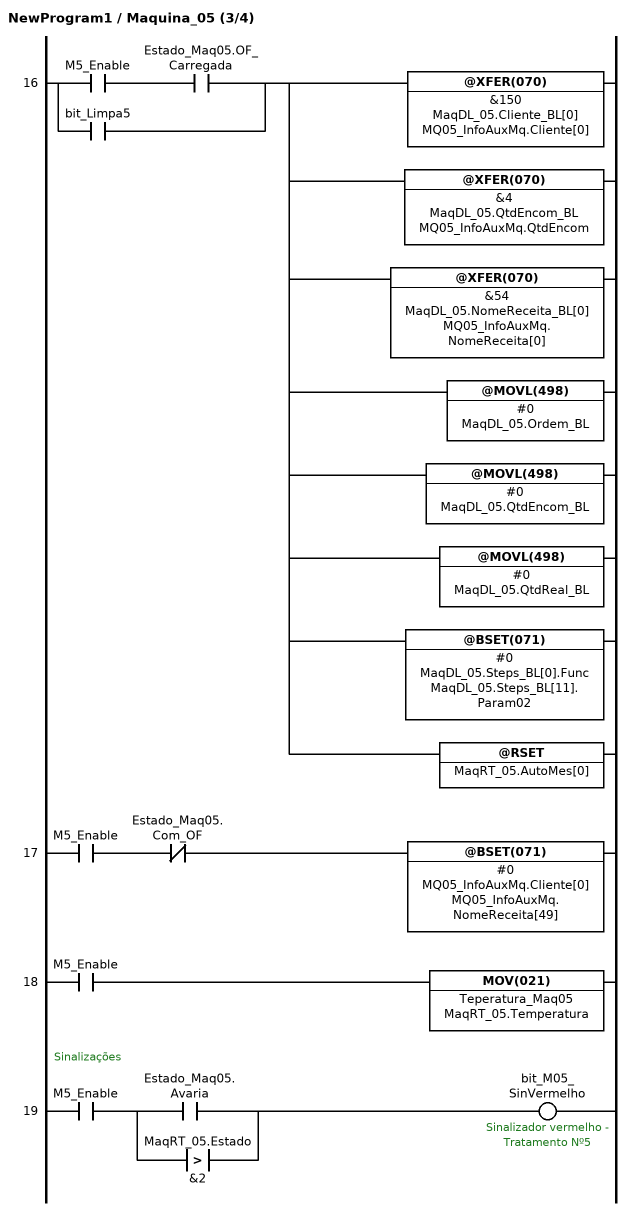
; rung 16
LD M5_Enable
AND Estado_Maq05.OF_Carregada
OR bit_Limpa5
@XFER(070) &150 MaqDL_05.Cliente_BL[0] MQ05_InfoAuxMq.Cliente[0]
@XFER(070) &4 MaqDL_05.QtdEncom_BL MQ05_InfoAuxMq.QtdEncom
@XFER(070) &54 MaqDL_05.NomeReceita_BL[0] MQ05_InfoAuxMq.NomeReceita[0]
@MOVL(498) #0 MaqDL_05.Ordem_BL
@MOVL(498) #0 MaqDL_05.QtdEncom_BL
@MOVL(498) #0 MaqDL_05.QtdReal_BL
@BSET(071) #0 MaqDL_05.Steps_BL[0].Func MaqDL_05.Steps_BL[11].Param02
@RSET MaqRT_05.AutoMes[0]
; rung 17
LD M5_Enable
ANDNOT Estado_Maq05.Com_OF
@BSET(071) #0 MQ05_InfoAuxMq.Cliente[0] MQ05_InfoAuxMq.NomeReceita[49]
; rung 18
LD M5_Enable
MOV(021) Teperatura_Maq05 MaqRT_05.Temperatura
; rung 19: Sinalizações
LD M5_Enable
LD Estado_Maq05.Avaria
OR>(320) MaqRT_05.Estado &2
ANDLD
OUT bit_M05_SinVermelho  ; Sinalizador vermelho - Tratamento Nº5

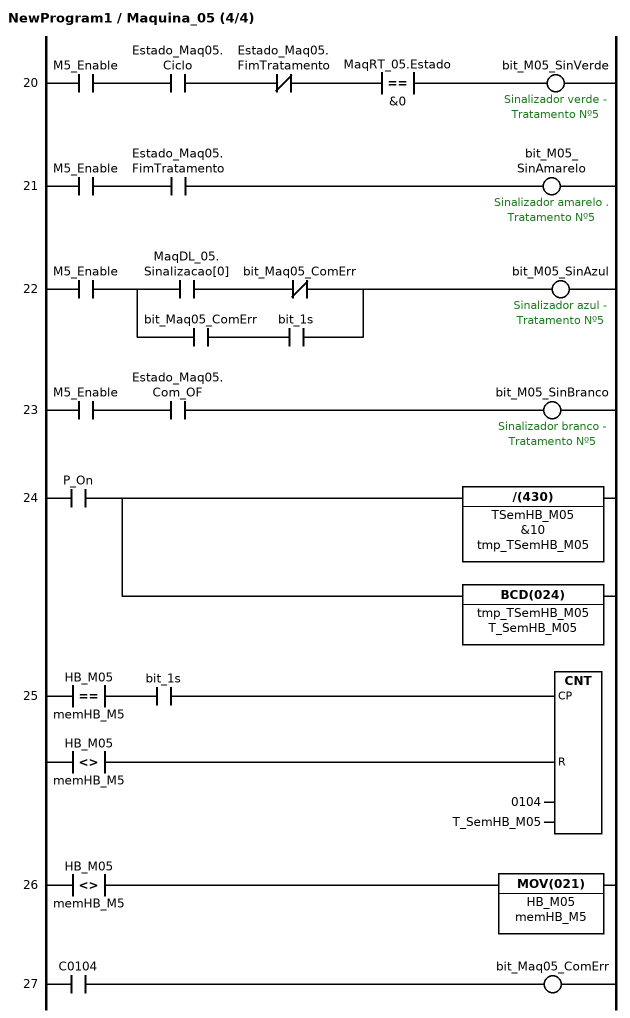
; rung 20
LD M5_Enable
AND Estado_Maq05.Ciclo
ANDNOT Estado_Maq05.FimTratamento
AND=(300) MaqRT_05.Estado &0
OUT bit_M05_SinVerde  ; Sinalizador verde - Tratamento Nº5
; rung 21
LD M5_Enable
AND Estado_Maq05.FimTratamento
OUT bit_M05_SinAmarelo  ; Sinalizador amarelo . Tratamento Nº5
; rung 22
LD M5_Enable
LD MaqDL_05.Sinalizacao[0]
ANDNOT bit_Maq05_ComErr
LD bit_Maq05_ComErr
AND bit_1s
ORLD
ANDLD
OUT bit_M05_SinAzul  ; Sinalizador azul - Tratamento Nº5
; rung 23
LD M5_Enable
AND Estado_Maq05.Com_OF
OUT bit_M05_SinBranco  ; Sinalizador branco - Tratamento Nº5
; rung 24
LD P_On
/(430) TSemHB_M05 &10 tmp_TSemHB_M05
BCD(024) tmp_TSemHB_M05 T_SemHB_M05
; rung 25
LD=(300) HB_M05 memHB_M5
AND bit_1s
LD<>(305) HB_M05 memHB_M5
CNT 0104 T_SemHB_M05
; rung 26
LD<>(305) HB_M05 memHB_M5
MOV(021) HB_M05 memHB_M5
; rung 27
LD C0104
OUT bit_Maq05_ComErr

### Section Maquina_06

